// TwinCAT 3 PLC project plc_lfe_gem
// Title: LFE GEM
// Company: SLAC - LCLS
// ProjectVersion: 4.0.0
// ProgramVersion: 3.1.4022.4
// libraries:
//   LCLS General, * (SLAC)
//   LCLS Vacuum, * (SLAC - LCLS)
//   PMPS, * (SLAC - LCLS)
//   Tc2_ControllerToolbox, * (Beckhoff Automation GmbH)
//   Tc2_Standard, * (Beckhoff Automation GmbH)
//   Tc2_System, * (Beckhoff Automation GmbH)
//   Tc2_Utilities, * (Beckhoff Automation GmbH)
//   Tc3_Module, * (Beckhoff Automation GmbH)
// project tree:
//   DUTs/ E_PositionState.TcDUT, ST_MPA.TcDUT, ST_PressureSensor.TcDUT
//   Version/ Global_Version.TcGVL
//   GVLs/ GVL_Control.TcGVL, GVL_Devices.TcGVL, GVL_ILK.TcGVL, GVL_Sensors.TcGVL
//   / PlcTask.TcTTO
//   POUs/ DIAGNOSTICS.TcPOU, FB_MPA.TcPOU, FB_PressureSensor_PX219.TcPOU, FB_VGC_1.TcPOU, MAIN.TcPOU, PRG_GEM1_DIFF_PUMP.TcPOU, PRG_GEM2_DIFF_PUMP.TcPOU, PRG_GATT.TcPOU, PRG_GEM1.TcPOU, PRG_GEM2.TcPOU, PRG_ILK.TcPOU, PRG_PMPS.TcPOU, PRG_ROOTS.TcPOU, PRG_SATT.TcPOU, PRG_SENSORS.TcPOU
// real-time tasks:
//   TASK PlcTask: cycle T#10ms, priority 20, ADS port 350
// I/O:
//   DEVICE EMxL0 (EtherCAT), AmsNetId 172.21.88.32.4.1
//     PLC_EMxL0 (EK1200) [EK1200-5000 EtherCAT Power supply (2A E-Bus)]
//       PLC_EL_1 (EL2088) [EL2088 8Ch. Dig. Output 24V, 0.5A, switching to negative]
//       PLC_EL_2 (EL1088) [EL1088 8Ch. Dig. Input 24V, 3ms, negative]
//       PLC_EL_3 (EL1088) [EL1088 8Ch. Dig. Input 24V, 3ms, negative]
//       PLC_EL_4 (EL3064) [EL3064 4Ch. Ana. Input 0-10V]
//       PLC_EL_5 (EL3064) [EL3064 4Ch. Ana. Input 0-10V]
//       PLC_EL_6 (EL2088) [EL2088 8Ch. Dig. Output 24V, 0.5A, switching to negative]
//       PLC_EL_7 (EL1088) [EL1088 8Ch. Dig. Input 24V, 3ms, negative]
//       PLC_EL_8 (EL1088) [EL1088 8Ch. Dig. Input 24V, 3ms, negative]
//       PLC_EL_9 (EL9187) [EL9187 Potential Connection, 8 x Ground]
//       PLC_EL_10 (EL2088) [EL2088 8Ch. Dig. Output 24V, 0.5A, switching to negative]
//       PLC_EL_11 (EL1088) [EL1088 8Ch. Dig. Input 24V, 3ms, negative]
//       PLC_EL_12 (EL1088) [EL1088 8Ch. Dig. Input 24V, 3ms, negative]
//       PLC_EL_13 (EL2088) [EL2088 8Ch. Dig. Output 24V, 0.5A, switching to negative]
//       PLC_EL_14 (EL9187) [EL9187 Potential Connection, 8 x Ground]
//       PLC_EL_15 (EL6070) [EL6070 1Ch. Licensing-Terminal]
//       PMPS_FFO [EL2202 2Ch. Dig. Output 24V, 0.5A]
//       PMPS_PRE [EL6692 EtherCAT Bridge terminal (Primary)]
//       PLC_EK_18 (EK1110) [EK1110 EtherCAT extension]
//     DRL_MKS (EK1100) [EK1100 EtherCAT Coupler (2A E-Bus)]
//       MKS_E1 (EL3064) [EL3064 4Ch. Ana. Input 0-10V]
//       MKS_E2 (EL3064) [EL3064 4Ch. Ana. Input 0-10V]
//       MKS_E3 (EL2794) [EL2794 4Ch. Dig. Output 24V AC/DC, 2A, short-circuit-proof]
//       MKS_E4 (EL3064) [EL3064 4Ch. Ana. Input 0-10V]
//       MKS_E5 (EL3064) [EL3064 4Ch. Ana. Input 0-10V]
//       MKS_E6 (EL2794) [EL2794 4Ch. Dig. Output 24V AC/DC, 2A, short-circuit-proof]
//       MKS_E7 (EL3064) [EL3064 4Ch. Ana. Input 0-10V]
//       MKS_E8 (EL3064) [EL3064 4Ch. Ana. Input 0-10V]
//       MKS_E9 (EL2794) [EL2794 4Ch. Dig. Output 24V AC/DC, 2A, short-circuit-proof]
//       MKS_E10 (EL3064) [EL3064 4Ch. Ana. Input 0-10V]
//       MKS_E11 (EL3064) [EL3064 4Ch. Ana. Input 0-10V]
//       MKS_E12 (EL2794) [EL2794 4Ch. Dig. Output 24V AC/DC, 2A, short-circuit-proof]
//       MKS_E13 (EL3064) [EL3064 4Ch. Ana. Input 0-10V]
//       MKS_E14 (EL3064) [EL3064 4Ch. Ana. Input 0-10V]
//       MKS_E15 (EL2794) [EL2794 4Ch. Dig. Output 24V AC/DC, 2A, short-circuit-proof]
//       MKS_E16 (EK1110)
//     DRL_PTM (EK1100) [EK1100 EtherCAT Coupler (2A E-Bus)]
//       PTM_E1_EL1004
//       PTM_E2_EL1004 [EL1004 4Ch. Dig. Input 24V, 3ms]
//       PTM_E3_EL2798 [EL2798 8Ch. Dig. Output 24V AC/DC, 2A, potential-free]
//       PTM_E4_EL3064 [EL3064 4Ch. Ana. Input 0-10V]
//       PTM_E5_EL4004 [EL4004 4Ch. Ana. Output 0-10V, 12bit]
//       PTM_E6_EL3064 [EL3064 4Ch. Ana. Input 0-10V]
//       PTM_E7_EL2798 [EL2798 8Ch. Dig. Output 24V AC/DC, 2A, potential-free]
//       PTM_E8_EL1004 [EL1004 4Ch. Dig. Input 24V, 3ms]
//       PTM_E9_EL1004
//       PTM_E10_EL9410
//       PTM_E11_EL1004
//       PTM_E12_EL1004 [EL1004 4Ch. Dig. Input 24V, 3ms]
//       PTM_E13_EL2798 [EL2798 8Ch. Dig. Output 24V AC/DC, 2A, potential-free]
//       PTM_E14_EL3064
//       PTM_E15_EL4004 [EL4004 4Ch. Ana. Output 0-10V, 12bit]
//       PTM_E16_EL3064 [EL3064 4Ch. Ana. Input 0-10V]
//       PTM_E17_EL2798 [EL2798 8Ch. Dig. Output 24V AC/DC, 2A, potential-free]
//       PTM_E18_EL1004
//       PTM_E19_EL1004 [EL1004 4Ch. Dig. Input 24V, 3ms]
//       PTM_E20_EL2624 [EL2624 4Ch. Relay Output, NO (125V AC / 30V DC)]
//       PTM_E21_EL1088 [EL1088 8Ch. Dig. Input 24V, 3ms, negative]
//       PTM_E22_EL9187 [EL9187 Potential Connection, 8 x Ground]
//       PTM_E23_EL9011
//     L0S3_PNL_01_EB_1 (EP2338-0002) [EP2338-0002 8 Ch. Dig. Input/Output 24V, 0,5A, M12]
//     L0S3_PNL_01_EB_2 (EP2338-0002) [EP2338-0002 8 Ch. Dig. Input/Output 24V, 0,5A, M12]
//     L0S3_PNL_01_EB_3 (EP2338-0002) [EP2338-0002 8 Ch. Dig. Input/Output 24V, 0,5A, M12]
//     L0S3_PNL_01_EB_4 (EP2338-0002) [EP2338-0002 8 Ch. Dig. Input/Output 24V, 0,5A, M12]
//     L0S3_PNL_01_EB_5 (EP3174-0002) [EP3174-0002 4Ch. Ana. Input +/-10V, 0-10V, 0/4-20mA configurable]
//     L0S3_PNL_01_EB_6 (EP3174-0002) [EP3174-0002 4Ch. Ana. Input +/-10V, 0-10V, 0/4-20mA configurable]
//     L0S3_PNL_02_EB_1 (EP2338-0002) [EP2338-0002 8 Ch. Dig. Input/Output 24V, 0,5A, M12]
//     L0S3_PNL_02_EB_2 (EP2338-0002) [EP2338-0002 8 Ch. Dig. Input/Output 24V, 0,5A, M12]
//     L0S3_PNL_02_EB_3 (EP4374-0002) [EP4374-0002 2Ch. Ana. Input +/-10V, 0-10V, 0/4-20mA configurable; 2Ch. Ana. Output +/-10V, 0-10V, 0/4-20mA configurable]
//     L0S3_PNL_02_EB_4 (EP3174-0002) [EP3174-0002 4Ch. Ana. Input +/-10V, 0-10V, 0/4-20mA configurable]
//     L0S3_PNL_02_EB_5 (EP2624-0002) [EP2624-0002 4Ch. Relay Output, NO (125V AC / 30V DC)]
//     L0S3_PNL_03_EB_1 (EP2338-0002) [EP2338-0002 8 Ch. Dig. Input/Output 24V, 0,5A, M12]
//     L0S3_PNL_03_EB_2 (EP2338-0002) [EP2338-0002 8 Ch. Dig. Input/Output 24V, 0,5A, M12]
//     L0S3_PNL_03_EB_3 (EP2338-0002) [EP2338-0002 8 Ch. Dig. Input/Output 24V, 0,5A, M12]
//     L0S3_PNL_03_EB_4 (EP3174-0002) [EP3174-0002 4Ch. Ana. Input +/-10V, 0-10V, 0/4-20mA configurable]
//     L0S3_PNL_03_EB_5 (EP3174-0002) [EP3174-0002 4Ch. Ana. Input +/-10V, 0-10V, 0/4-20mA configurable]
//     L0S3_PNL_03_EB_6 (EP2624-0002) [EP2624-0002 4Ch. Relay Output, NO (125V AC / 30V DC)]
//     L0S3_PNL_03_EB_7 (EP2338-0002) [EP2338-0002 8 Ch. Dig. Input/Output 24V, 0,5A, M12]
//     L0S3_PNL_03_EB_8 (EP2624-0002) [EP2624-0002 4Ch. Relay Output, NO (125V AC / 30V DC)]
//     L0S3_PNL_03_EB_9 (EP2338-0002) [EP2338-0002 8 Ch. Dig. Input/Output 24V, 0,5A, M12]
//     L0S6_PNL_04_EB_1 (EP2338-0002) [EP2338-0002 8 Ch. Dig. Input/Output 24V, 0,5A, M12]
//     L0S6_PNL_04_EB_2 (EP3174-0002) [EP3174-0002 4Ch. Ana. Input +/-10V, 0-10V, 0/4-20mA configurable]
//     L0S6_PNL_04_EB_3 (EP4374-0002) [EP4374-0002 2Ch. Ana. Input +/-10V, 0-10V, 0/4-20mA configurable; 2Ch. Ana. Output +/-10V, 0-10V, 0/4-20mA configurable]
//     L0S6_PNL_04_EB_4 (EP2338-0002) [EP2338-0002 8 Ch. Dig. Input/Output 24V, 0,5A, M12]
//     L0S6_PNL_04_EB_5 (EP2338-0002) [EP2338-0002 8 Ch. Dig. Input/Output 24V, 0,5A, M12]
//     L0S6_PNL_04_EB_6 (EP2338-0002) [EP2338-0002 8 Ch. Dig. Input/Output 24V, 0,5A, M12]
//     L0S6_PNL_04_EB_7 (EP2338-0002) [EP2338-0002 8 Ch. Dig. Input/Output 24V, 0,5A, M12]
//     L0S6_PNL_04_EB_8 (EP2338-0002) [EP2338-0002 8 Ch. Dig. Input/Output 24V, 0,5A, M12]
//     L0S6_PNL_01_EB_1 (EP2338-0002) [EP2338-0002 8 Ch. Dig. Input/Output 24V, 0,5A, M12]
//     L0S6_PNL_01_EB_2 (EP2338-0002) [EP2338-0002 8 Ch. Dig. Input/Output 24V, 0,5A, M12]
//     L0S6_PNL_01_EB_3 (EP2338-0002) [EP2338-0002 8 Ch. Dig. Input/Output 24V, 0,5A, M12]
//     L0S6_PNL_01_EB_4 (EP3174-0002) [EP3174-0002 4Ch. Ana. Input +/-10V, 0-10V, 0/4-20mA configurable]
//     L0S6_PNL_01_EB_5 (EP3174-0002) [EP3174-0002 4Ch. Ana. Input +/-10V, 0-10V, 0/4-20mA configurable]
//     L0S6_PNL_01_EB_6 (EP2624-0002) [EP2624-0002 4Ch. Relay Output, NO (125V AC / 30V DC)]
//     L0S6_PNL_01_EB_7 (EP2338-0002) [EP2338-0002 8 Ch. Dig. Input/Output 24V, 0,5A, M12]
//     L0S6_PNL_01_EB_8 (EP2624-0002) [EP2624-0002 4Ch. Relay Output, NO (125V AC / 30V DC)]
//     L0S6_PNL_01_EB_9 (EP2338-0002) [EP2338-0002 8 Ch. Dig. Input/Output 24V, 0,5A, M12]
//     L0S6_PNL_02_EB_1 (EP2338-0002) [EP2338-0002 8 Ch. Dig. Input/Output 24V, 0,5A, M12]
//     L0S6_PNL_02_EB_2 (EP2338-0002) [EP2338-0002 8 Ch. Dig. Input/Output 24V, 0,5A, M12]
//     L0S6_PNL_02_EB_3 (EP4374-0002) [EP4374-0002 2Ch. Ana. Input +/-10V, 0-10V, 0/4-20mA configurable; 2Ch. Ana. Output +/-10V, 0-10V, 0/4-20mA configurable]
//     L0S6_PNL_02_EB_4 (EP3174-0002) [EP3174-0002 4Ch. Ana. Input +/-10V, 0-10V, 0/4-20mA configurable]
//     L0S6_PNL_02_EB_5 (EP2624-0002) [EP2624-0002 4Ch. Relay Output, NO (125V AC / 30V DC)]
//     L0S6_PNL_03_EB_1 (EP2338-0002) [EP2338-0002 8 Ch. Dig. Input/Output 24V, 0,5A, M12]
//     L0S6_PNL_03_EB_2 (EP2338-0002) [EP2338-0002 8 Ch. Dig. Input/Output 24V, 0,5A, M12]
//     L0S6_PNL_03_EB_3 (EP2338-0002) [EP2338-0002 8 Ch. Dig. Input/Output 24V, 0,5A, M12]
//     L0S6_PNL_03_EB_4 (EP2338-0002) [EP2338-0002 8 Ch. Dig. Input/Output 24V, 0,5A, M12]
//     L0S6_PNL_03_EB_5 (EP3174-0002) [EP3174-0002 4Ch. Ana. Input +/-10V, 0-10V, 0/4-20mA configurable]
//     L0S6_PNL_03_EB_6 (EP3174-0002) [EP3174-0002 4Ch. Ana. Input +/-10V, 0-10V, 0/4-20mA configurable]
// variable links:
//   plc_lfe_gem/plc_lfe_gem Instance <-> EMxL0 (EtherCAT)/DRL_MKS (EK1100)/MKS_E1 (EL3064)
//     PlcTask Inputs/GVL_Devices.GEM1_GCC_10.i_iPRESS_R <-> AI Standard Channel 1/Value
//     PlcTask Inputs/GVL_Devices.GEM1_GCC_20.i_iPRESS_R <-> AI Standard Channel 3/Value
//     PlcTask Inputs/GVL_Devices.GEM1_GPI_10.i_iPRESS_R <-> AI Standard Channel 4/Value
//   plc_lfe_gem/plc_lfe_gem Instance <-> EMxL0 (EtherCAT)/DRL_MKS (EK1100)/MKS_E10 (EL3064)
//     PlcTask Inputs/GVL_Devices.GEM2_GCC_50.i_iPRESS_R <-> AI Standard Channel 1/Value
//     PlcTask Inputs/GVL_Devices.GEM2_GCC_60.i_iPRESS_R <-> AI Standard Channel 3/Value
//     PlcTask Inputs/GVL_Devices.GEM2_GPI_50.i_iPRESS_R <-> AI Standard Channel 4/Value
//   plc_lfe_gem/plc_lfe_gem Instance <-> EMxL0 (EtherCAT)/DRL_MKS (EK1100)/MKS_E11 (EL3064)
//     PlcTask Inputs/GVL_Devices.GEM2_GPI_60.i_iPRESS_R <-> AI Standard Channel 1/Value
//   plc_lfe_gem/plc_lfe_gem Instance <-> EMxL0 (EtherCAT)/DRL_MKS (EK1100)/MKS_E12 (EL2794)
//     PlcTask Outputs/GVL_Devices.GEM2_GCC_50.q_xHV_DIS <-> Channel 1/Output
//     PlcTask Outputs/GVL_Devices.GEM2_GCC_60.q_xHV_DIS <-> Channel 2/Output
//   plc_lfe_gem/plc_lfe_gem Instance <-> EMxL0 (EtherCAT)/DRL_MKS (EK1100)/MKS_E13 (EL3064)
//     PlcTask Inputs/GVL_Devices.GEM2_GCC_70.i_iPRESS_R <-> AI Standard Channel 1/Value
//     PlcTask Inputs/GVL_Devices.GEM2_GPI_70.i_iPRESS_R <-> AI Standard Channel 4/Value
//   plc_lfe_gem/plc_lfe_gem Instance <-> EMxL0 (EtherCAT)/DRL_MKS (EK1100)/MKS_E14 (EL3064)
//     PlcTask Inputs/GVL_Devices.GEM1_GPI_60.i_iPRESS_R <-> AI Standard Channel 1/Value
//   plc_lfe_gem/plc_lfe_gem Instance <-> EMxL0 (EtherCAT)/DRL_MKS (EK1100)/MKS_E15 (EL2794)
//     PlcTask Outputs/GVL_Devices.GEM2_GCC_70.q_xHV_DIS <-> Channel 1/Output
//   plc_lfe_gem/plc_lfe_gem Instance <-> EMxL0 (EtherCAT)/DRL_MKS (EK1100)/MKS_E2 (EL3064)
//     PlcTask Inputs/GVL_Devices.GEM1_GPI_20.i_iPRESS_R <-> AI Standard Channel 1/Value
//   plc_lfe_gem/plc_lfe_gem Instance <-> EMxL0 (EtherCAT)/DRL_MKS (EK1100)/MKS_E3 (EL2794)
//     PlcTask Outputs/GVL_Devices.GEM1_GCC_10.q_xHV_DIS <-> Channel 1/Output
//     PlcTask Outputs/GVL_Devices.GEM1_GCC_20.q_xHV_DIS <-> Channel 2/Output
//   plc_lfe_gem/plc_lfe_gem Instance <-> EMxL0 (EtherCAT)/DRL_MKS (EK1100)/MKS_E4 (EL3064)
//     PlcTask Inputs/GVL_Devices.GEM1_GCC_30.i_iPRESS_R <-> AI Standard Channel 1/Value
//     PlcTask Inputs/GVL_Devices.GEM1_GCC_50.i_iPRESS_R <-> AI Standard Channel 3/Value
//     PlcTask Inputs/GVL_Devices.GEM1_GPI_30.i_iPRESS_R <-> AI Standard Channel 4/Value
//   plc_lfe_gem/plc_lfe_gem Instance <-> EMxL0 (EtherCAT)/DRL_MKS (EK1100)/MKS_E5 (EL3064)
//     PlcTask Inputs/GVL_Devices.GEM1_GPI_50.i_iPRESS_R <-> AI Standard Channel 1/Value
//   plc_lfe_gem/plc_lfe_gem Instance <-> EMxL0 (EtherCAT)/DRL_MKS (EK1100)/MKS_E6 (EL2794)
//     PlcTask Outputs/GVL_Devices.GEM1_GCC_30.q_xHV_DIS <-> Channel 1/Output
//     PlcTask Outputs/GVL_Devices.GEM1_GCC_50.q_xHV_DIS <-> Channel 2/Output
//   plc_lfe_gem/plc_lfe_gem Instance <-> EMxL0 (EtherCAT)/DRL_MKS (EK1100)/MKS_E7 (EL3064)
//     PlcTask Inputs/GVL_Devices.GATT_GPI_10.i_iPRESS_R <-> AI Standard Channel 2/Value
//     PlcTask Inputs/GVL_Devices.GEM2_GCC_30.i_iPRESS_R <-> AI Standard Channel 1/Value
//     PlcTask Inputs/GVL_Devices.GEM2_GPI_10.i_iPRESS_R <-> AI Standard Channel 4/Value
//     PlcTask Inputs/GVL_Devices.GEM2_GPI_30.i_iPRESS_R <-> AI Standard Channel 3/Value
//   plc_lfe_gem/plc_lfe_gem Instance <-> EMxL0 (EtherCAT)/DRL_MKS (EK1100)/MKS_E9 (EL2794)
//     PlcTask Outputs/GVL_Devices.GEM2_GCC_30.q_xHV_DIS <-> Channel 1/Output
//   plc_lfe_gem/plc_lfe_gem Instance <-> EMxL0 (EtherCAT)/DRL_PTM (EK1100)/PTM_E11_EL1004
//     PlcTask Inputs/GVL_Devices.GEM2_PTM_30.i_xAtSpd <-> Channel 2/Input
//     PlcTask Inputs/GVL_Devices.GEM2_PTM_30.i_xDecel <-> Channel 1/Input
//     PlcTask Inputs/GVL_Devices.GEM2_PTM_30.i_xNCFault <-> Channel 3/Input
//     PlcTask Inputs/GVL_Devices.GEM2_PTM_30.i_xRotate <-> Channel 4/Input
//   plc_lfe_gem/plc_lfe_gem Instance <-> EMxL0 (EtherCAT)/DRL_PTM (EK1100)/PTM_E12_EL1004
//     PlcTask Inputs/GVL_Devices.GEM2_PTM_30.i_xAccel <-> Channel 1/Input
//   plc_lfe_gem/plc_lfe_gem Instance <-> EMxL0 (EtherCAT)/DRL_PTM (EK1100)/PTM_E13_EL2798
//     PlcTask Outputs/GVL_Devices.GEM2_PTM_30.q_xProtection <-> Channel 4/Output
//     PlcTask Outputs/GVL_Devices.GEM2_PTM_30.q_xReset <-> Channel 1/Output
//     PlcTask Outputs/GVL_Devices.GEM2_PTM_30.q_xSetSpeed <-> Channel 5/Output
//     PlcTask Outputs/GVL_Devices.GEM2_PTM_30.q_xStart <-> Channel 2/Output
//     PlcTask Outputs/GVL_Devices.GEM2_PTM_30.q_xStop <-> Channel 3/Output
//   plc_lfe_gem/plc_lfe_gem Instance <-> EMxL0 (EtherCAT)/DRL_PTM (EK1100)/PTM_E14_EL3064
//     PlcTask Inputs/GVL_Devices.GEM2_PTM_30.i_iCurrentMon <-> AI Standard Channel 2/Value
//     PlcTask Inputs/GVL_Devices.GEM2_PTM_30.i_iRawSpeed <-> AI Standard Channel 1/Value
//     PlcTask Inputs/GVL_Devices.GEM2_PTM_30.i_iTempMon <-> AI Standard Channel 3/Value
//   plc_lfe_gem/plc_lfe_gem Instance <-> EMxL0 (EtherCAT)/DRL_PTM (EK1100)/PTM_E15_EL4004
//     PlcTask Outputs/GVL_Devices.GEM2_PTM_30.q_iSpeedSet <-> AO Outputs Channel 1/Analog output
//     PlcTask Outputs/GVL_Devices.GEM2_PTM_50.q_iSpeedSet <-> AO Outputs Channel 3/Analog output
//   plc_lfe_gem/plc_lfe_gem Instance <-> EMxL0 (EtherCAT)/DRL_PTM (EK1100)/PTM_E16_EL3064
//     PlcTask Inputs/GVL_Devices.GEM2_PTM_50.i_iCurrentMon <-> AI Standard Channel 2/Value
//     PlcTask Inputs/GVL_Devices.GEM2_PTM_50.i_iRawSpeed <-> AI Standard Channel 1/Value
//     PlcTask Inputs/GVL_Devices.GEM2_PTM_50.i_iTempMon <-> AI Standard Channel 3/Value
//   plc_lfe_gem/plc_lfe_gem Instance <-> EMxL0 (EtherCAT)/DRL_PTM (EK1100)/PTM_E17_EL2798
//     PlcTask Outputs/GVL_Devices.GEM2_PTM_50.q_xProtection <-> Channel 4/Output
//     PlcTask Outputs/GVL_Devices.GEM2_PTM_50.q_xReset <-> Channel 1/Output
//     PlcTask Outputs/GVL_Devices.GEM2_PTM_50.q_xSetSpeed <-> Channel 5/Output
//     PlcTask Outputs/GVL_Devices.GEM2_PTM_50.q_xStart <-> Channel 2/Output
//     PlcTask Outputs/GVL_Devices.GEM2_PTM_50.q_xStop <-> Channel 3/Output
//   plc_lfe_gem/plc_lfe_gem Instance <-> EMxL0 (EtherCAT)/DRL_PTM (EK1100)/PTM_E18_EL1004
//     PlcTask Inputs/GVL_Devices.GEM2_PTM_50.i_xAtSpd <-> Channel 2/Input
//     PlcTask Inputs/GVL_Devices.GEM2_PTM_50.i_xDecel <-> Channel 1/Input
//     PlcTask Inputs/GVL_Devices.GEM2_PTM_50.i_xNCFault <-> Channel 3/Input
//     PlcTask Inputs/GVL_Devices.GEM2_PTM_50.i_xRotate <-> Channel 4/Input
//   plc_lfe_gem/plc_lfe_gem Instance <-> EMxL0 (EtherCAT)/DRL_PTM (EK1100)/PTM_E19_EL1004
//     PlcTask Inputs/GVL_Devices.GEM2_PTM_50.i_xAccel <-> Channel 1/Input
//   plc_lfe_gem/plc_lfe_gem Instance <-> EMxL0 (EtherCAT)/DRL_PTM (EK1100)/PTM_E1_EL1004
//     PlcTask Inputs/GVL_Devices.GEM1_PTM_30.i_xAtSpd <-> Channel 2/Input
//     PlcTask Inputs/GVL_Devices.GEM1_PTM_30.i_xDecel <-> Channel 1/Input
//     PlcTask Inputs/GVL_Devices.GEM1_PTM_30.i_xNCFault <-> Channel 3/Input
//     PlcTask Inputs/GVL_Devices.GEM1_PTM_30.i_xRotate <-> Channel 4/Input
//   plc_lfe_gem/plc_lfe_gem Instance <-> EMxL0 (EtherCAT)/DRL_PTM (EK1100)/PTM_E20_EL2624
//     PlcTask Outputs/GVL_Devices.GEM1_PTM_10.q_RunDO <-> Channel 1/Output
//     PlcTask Outputs/GVL_Devices.GEM1_PTM_20.q_RunDO <-> Channel 2/Output
//     PlcTask Outputs/GVL_Devices.GEM2_PTM_60.q_RunDO <-> Channel 3/Output
//     PlcTask Outputs/GVL_Devices.GEM2_PTM_70.q_RunDO <-> Channel 4/Output
//   plc_lfe_gem/plc_lfe_gem Instance <-> EMxL0 (EtherCAT)/DRL_PTM (EK1100)/PTM_E21_EL1088
//     PlcTask Inputs/GVL_Devices.GEM1_PTM_10.i_xAtSpd <-> Channel 1/Input
//     PlcTask Inputs/GVL_Devices.GEM1_PTM_20.i_xAtSpd <-> Channel 3/Input
//     PlcTask Inputs/GVL_Devices.GEM2_PTM_60.i_xAtSpd <-> Channel 5/Input
//     PlcTask Inputs/GVL_Devices.GEM2_PTM_70.i_xAtSpd <-> Channel 7/Input
//     PlcTask Inputs/GVL_Devices.GEM1_PTM_10.i_xFault <-> Channel 2/Input
//     PlcTask Inputs/GVL_Devices.GEM1_PTM_20.i_xFault <-> Channel 4/Input
//     PlcTask Inputs/GVL_Devices.GEM2_PTM_60.i_xFault <-> Channel 6/Input
//     PlcTask Inputs/GVL_Devices.GEM2_PTM_70.i_xFault <-> Channel 8/Input
//   plc_lfe_gem/plc_lfe_gem Instance <-> EMxL0 (EtherCAT)/DRL_PTM (EK1100)/PTM_E2_EL1004
//     PlcTask Inputs/GVL_Devices.GEM1_PTM_30.i_xAccel <-> Channel 1/Input
//   plc_lfe_gem/plc_lfe_gem Instance <-> EMxL0 (EtherCAT)/DRL_PTM (EK1100)/PTM_E3_EL2798
//     PlcTask Outputs/GVL_Devices.GEM1_PTM_30.q_xProtection <-> Channel 4/Output
//     PlcTask Outputs/GVL_Devices.GEM1_PTM_30.q_xReset <-> Channel 1/Output
//     PlcTask Outputs/GVL_Devices.GEM1_PTM_30.q_xSetSpeed <-> Channel 5/Output
//     PlcTask Outputs/GVL_Devices.GEM1_PTM_30.q_xStart <-> Channel 2/Output
//     PlcTask Outputs/GVL_Devices.GEM1_PTM_30.q_xStop <-> Channel 3/Output
//   plc_lfe_gem/plc_lfe_gem Instance <-> EMxL0 (EtherCAT)/DRL_PTM (EK1100)/PTM_E4_EL3064
//     PlcTask Inputs/GVL_Devices.GEM1_PTM_30.i_iCurrentMon <-> AI Standard Channel 2/Value
//     PlcTask Inputs/GVL_Devices.GEM1_PTM_30.i_iRawSpeed <-> AI Standard Channel 1/Value
//     PlcTask Inputs/GVL_Devices.GEM1_PTM_30.i_iTempMon <-> AI Standard Channel 3/Value
//   plc_lfe_gem/plc_lfe_gem Instance <-> EMxL0 (EtherCAT)/DRL_PTM (EK1100)/PTM_E5_EL4004
//     PlcTask Outputs/GVL_Devices.GEM1_PTM_30.q_iSpeedSet <-> AO Outputs Channel 1/Analog output
//     PlcTask Outputs/GVL_Devices.GEM1_PTM_50.q_iSpeedSet <-> AO Outputs Channel 3/Analog output
//   plc_lfe_gem/plc_lfe_gem Instance <-> EMxL0 (EtherCAT)/DRL_PTM (EK1100)/PTM_E6_EL3064
//     PlcTask Inputs/GVL_Devices.GEM1_PTM_50.i_iCurrentMon <-> AI Standard Channel 2/Value
//     PlcTask Inputs/GVL_Devices.GEM1_PTM_50.i_iRawSpeed <-> AI Standard Channel 1/Value
//     PlcTask Inputs/GVL_Devices.GEM1_PTM_50.i_iTempMon <-> AI Standard Channel 3/Value
//   plc_lfe_gem/plc_lfe_gem Instance <-> EMxL0 (EtherCAT)/DRL_PTM (EK1100)/PTM_E7_EL2798
//     PlcTask Outputs/GVL_Devices.GEM1_PTM_50.q_xProtection <-> Channel 4/Output
//     PlcTask Outputs/GVL_Devices.GEM1_PTM_50.q_xReset <-> Channel 1/Output
//     PlcTask Outputs/GVL_Devices.GEM1_PTM_50.q_xSetSpeed <-> Channel 5/Output
//     PlcTask Outputs/GVL_Devices.GEM1_PTM_50.q_xStart <-> Channel 2/Output
//     PlcTask Outputs/GVL_Devices.GEM1_PTM_50.q_xStop <-> Channel 3/Output
//   plc_lfe_gem/plc_lfe_gem Instance <-> EMxL0 (EtherCAT)/DRL_PTM (EK1100)/PTM_E8_EL1004
//     PlcTask Inputs/GVL_Devices.GEM1_PTM_50.i_xAtSpd <-> Channel 2/Input
//     PlcTask Inputs/GVL_Devices.GEM1_PTM_50.i_xDecel <-> Channel 1/Input
//     PlcTask Inputs/GVL_Devices.GEM1_PTM_50.i_xNCFault <-> Channel 3/Input
//     PlcTask Inputs/GVL_Devices.GEM1_PTM_50.i_xRotate <-> Channel 4/Input
//   plc_lfe_gem/plc_lfe_gem Instance <-> EMxL0 (EtherCAT)/DRL_PTM (EK1100)/PTM_E9_EL1004
//     PlcTask Inputs/GVL_Devices.GEM1_PTM_50.i_xAccel <-> Channel 1/Input
//   plc_lfe_gem/plc_lfe_gem Instance <-> EMxL0 (EtherCAT)/L0S3_PNL_01_EB_1 (EP2338-0002)
//     PlcTask Inputs/GVL_Devices.GEM1_VGC_10.i_xClsLS <-> Channel 2/Input
//     PlcTask Inputs/GVL_Devices.GEM1_VGC_10.i_xOpnLS <-> Channel 1/Input
//     PlcTask Inputs/GVL_Devices.GEM1_VRC_10.i_xClsLS <-> Channel 6/Input
//     PlcTask Inputs/GVL_Devices.GEM1_VRC_10.i_xOpnLS <-> Channel 5/Input
//     PlcTask Outputs/GVL_Devices.GEM1_VGC_10.q_xOPN_DO <-> Channel 11/Output
//     PlcTask Outputs/GVL_Devices.GEM1_VRC_10.q_xOPN_DO <-> Channel 15/Output
//   plc_lfe_gem/plc_lfe_gem Instance <-> EMxL0 (EtherCAT)/L0S3_PNL_01_EB_2 (EP2338-0002)
//     PlcTask Inputs/GVL_Devices.GEM1_VGC_20.i_xClsLS <-> Channel 2/Input
//     PlcTask Inputs/GVL_Devices.GEM1_VGC_30.i_xClsLS <-> Channel 6/Input
//     PlcTask Inputs/GVL_Devices.GEM1_VGC_20.i_xOpnLS <-> Channel 1/Input
//     PlcTask Inputs/GVL_Devices.GEM1_VGC_30.i_xOpnLS <-> Channel 5/Input
//     PlcTask Outputs/GVL_Devices.GEM1_VGC_20.q_xOPN_DO <-> Channel 11/Output
//     PlcTask Outputs/GVL_Devices.GEM1_VGC_30.q_xOPN_DO <-> Channel 15/Output
//   plc_lfe_gem/plc_lfe_gem Instance <-> EMxL0 (EtherCAT)/L0S3_PNL_01_EB_3 (EP2338-0002)
//     PlcTask Inputs/GVL_Devices.GEM1_VRC_20.i_xClsLS <-> Channel 6/Input
//     PlcTask Inputs/GVL_Devices.GEM1_VRC_20.i_xOpnLS <-> Channel 5/Input
//     PlcTask Outputs/GVL_Devices.GEM1_VRC_20.q_xOPN_DO <-> Channel 15/Output
//     PlcTask Outputs/GVL_Devices.GEM1_VVC_20.q_xCLS_DO <-> Channel 11/Output
//   plc_lfe_gem/plc_lfe_gem Instance <-> EMxL0 (EtherCAT)/L0S3_PNL_01_EB_4 (EP2338-0002)
//     PlcTask Inputs/GVL_Devices.GEM1_VRC_30.i_xClsLS <-> Channel 6/Input
//     PlcTask Inputs/GVL_Devices.GEM1_VRC_30.i_xOpnLS <-> Channel 5/Input
//     PlcTask Outputs/GVL_Devices.GEM1_VRC_30.q_xOPN_DO <-> Channel 15/Output
//     PlcTask Outputs/GVL_Devices.GEM1_VVC_30.q_xCLS_DO <-> Channel 11/Output
//   plc_lfe_gem/plc_lfe_gem Instance <-> EMxL0 (EtherCAT)/L0S3_PNL_01_EB_5 (EP3174-0002)
//     PlcTask Inputs/GVL_Devices.GEM1_GPI_11.i_iPRESS_R <-> AI Standard Channel 3/Value
//     PlcTask Inputs/GVL_Devices.GEM1_GPI_31.i_iPRESS_R <-> AI Standard Channel 4/Value
//   plc_lfe_gem/plc_lfe_gem Instance <-> EMxL0 (EtherCAT)/L0S3_PNL_02_EB_1 (EP2338-0002)
//     PlcTask Inputs/GVL_Devices.GEM1_VGC_40.i_xClsLS <-> Channel 2/Input
//     PlcTask Inputs/GVL_Devices.GEM1_VGC_50.i_xClsLS <-> Channel 6/Input
//     PlcTask Inputs/GVL_Devices.GEM1_VGC_40.i_xOpnLS <-> Channel 1/Input
//     PlcTask Inputs/GVL_Devices.GEM1_VGC_50.i_xOpnLS <-> Channel 5/Input
//     PlcTask Outputs/GVL_Devices.GEM1_VGC_40.q_xOPN_DO <-> Channel 11/Output
//     PlcTask Outputs/GVL_Devices.GEM1_VGC_50.q_xOPN_DO <-> Channel 15/Output
//   plc_lfe_gem/plc_lfe_gem Instance <-> EMxL0 (EtherCAT)/L0S3_PNL_02_EB_2 (EP2338-0002)
//     PlcTask Outputs/GVL_Devices.GEM1_VVC_40.q_xOPN_DO <-> Channel 15/Output
//   plc_lfe_gem/plc_lfe_gem Instance <-> EMxL0 (EtherCAT)/L0S3_PNL_02_EB_3 (EP4374-0002)
//     PlcTask Outputs/GVL_Devices.GEM1_VCN_40.q_iRawPosition <-> AO Outputs Channel 4/Analog output
//   plc_lfe_gem/plc_lfe_gem Instance <-> EMxL0 (EtherCAT)/L0S3_PNL_02_EB_4 (EP3174-0002)
//     PlcTask Inputs/GVL_Devices.GEM1_GCM_41.i_iPRESS_R <-> AI Standard Channel 1/Value
//     PlcTask Inputs/GVL_Devices.GEM1_GCM_42.i_iPRESS_R <-> AI Standard Channel 2/Value
//   plc_lfe_gem/plc_lfe_gem Instance <-> EMxL0 (EtherCAT)/L0S3_PNL_03_EB_1 (EP2338-0002)
//     PlcTask Inputs/GVL_Devices.GEM1_VGC_60.i_xClsLS <-> Channel 6/Input
//     PlcTask Inputs/GVL_Devices.GEM1_VGC_60.i_xOpnLS <-> Channel 5/Input
//     PlcTask Inputs/GVL_Devices.GEM1_VRC_50.i_xClsLS <-> Channel 2/Input
//     PlcTask Inputs/GVL_Devices.GEM1_VRC_50.i_xOpnLS <-> Channel 1/Input
//     PlcTask Outputs/GVL_Devices.GEM1_VGC_60.q_xOPN_DO <-> Channel 15/Output
//     PlcTask Outputs/GVL_Devices.GEM1_VRC_50.q_xOPN_DO <-> Channel 11/Output
//   plc_lfe_gem/plc_lfe_gem Instance <-> EMxL0 (EtherCAT)/L0S3_PNL_03_EB_2 (EP2338-0002)
//     PlcTask Inputs/GVL_Devices.GEM1_VRC_60.i_xClsLS <-> Channel 6/Input
//     PlcTask Inputs/GVL_Devices.GEM1_VRC_60.i_xOpnLS <-> Channel 5/Input
//     PlcTask Outputs/GVL_Devices.GEM1_VRC_60.q_xOPN_DO <-> Channel 15/Output
//     PlcTask Outputs/GVL_Devices.GEM1_VVC_50.q_xCLS_DO <-> Channel 11/Output
//   plc_lfe_gem/plc_lfe_gem Instance <-> EMxL0 (EtherCAT)/L0S3_PNL_03_EB_3 (EP2338-0002)
//     PlcTask Inputs/GVL_Devices.GEM1_VGC_70.i_xClsLS <-> Channel 2/Input
//     PlcTask Inputs/GVL_Devices.GEM1_VGC_70.i_xOpnLS <-> Channel 1/Input
//     PlcTask Inputs/GVL_Devices.GEM1_VRC_70.i_xClsLS <-> Channel 6/Input
//     PlcTask Inputs/GVL_Devices.GEM1_VRC_70.i_xOpnLS <-> Channel 5/Input
//     PlcTask Outputs/GVL_Devices.GEM1_VGC_70.q_xOPN_DO <-> Channel 11/Output
//     PlcTask Outputs/GVL_Devices.GEM1_VRC_70.q_xOPN_DO <-> Channel 15/Output
//   plc_lfe_gem/plc_lfe_gem Instance <-> EMxL0 (EtherCAT)/L0S3_PNL_03_EB_4 (EP3174-0002)
//     PlcTask Inputs/GVL_Devices.GEM1_GPI_51.i_iPRESS_R <-> AI Standard Channel 3/Value
//   plc_lfe_gem/plc_lfe_gem Instance <-> EMxL0 (EtherCAT)/L0S3_PNL_03_EB_5 (EP3174-0002)
//     PlcTask Inputs/GVL_Devices.GEM1_GPI_61.i_iPRESS_R <-> AI Standard Channel 2/Value
//     PlcTask Inputs/GVL_Devices.GEM1_GPI_71.i_iPRESS_R <-> AI Standard Channel 3/Value
//   plc_lfe_gem/plc_lfe_gem Instance <-> EMxL0 (EtherCAT)/L0S3_PNL_03_EB_6 (EP2624-0002)
//     PlcTask Outputs/GVL_Devices.GEM1_PRO_60.q_xLspdDo <-> Channel 2/Output
//     PlcTask Outputs/GVL_Devices.GEM1_PRO_60.q_xResetDo <-> Channel 3/Output
//     PlcTask Outputs/GVL_Devices.GEM1_PRO_60.q_xRunDO <-> Channel 1/Output
//   plc_lfe_gem/plc_lfe_gem Instance <-> EMxL0 (EtherCAT)/L0S3_PNL_03_EB_7 (EP2338-0002)
//     PlcTask Inputs/GVL_Devices.GEM1_PRO_60.i_xAlarm <-> Channel 6/Input
//     PlcTask Inputs/GVL_Devices.GEM1_PRO_60.i_xIsRun <-> Channel 1/Input
//     PlcTask Inputs/GVL_Devices.GEM1_PRO_60.i_xWarning <-> Channel 5/Input
//     PlcTask Outputs/GVL_Devices.GEM1_PRO_20.q_xRunDo <-> Channel 11/Output
//     PlcTask Outputs/GVL_Devices.GEM1_PRO_30.q_xRunDo <-> Channel 12/Output
//     PlcTask Outputs/GVL_Devices.GEM1_PRO_50.q_xRunDo <-> Channel 15/Output
//   plc_lfe_gem/plc_lfe_gem Instance <-> EMxL0 (EtherCAT)/L0S3_PNL_03_EB_8 (EP2624-0002)
//     PlcTask Outputs/GVL_Devices.GEM1_PRO_70.q_xLspdDo <-> Channel 2/Output
//     PlcTask Outputs/GVL_Devices.GEM1_PRO_70.q_xResetDo <-> Channel 3/Output
//     PlcTask Outputs/GVL_Devices.GEM1_PRO_70.q_xRunDO <-> Channel 1/Output
//   plc_lfe_gem/plc_lfe_gem Instance <-> EMxL0 (EtherCAT)/L0S3_PNL_03_EB_9 (EP2338-0002)
//     PlcTask Inputs/GVL_Devices.GEM1_PRO_70.i_xAlarm <-> Channel 6/Input
//     PlcTask Inputs/GVL_Devices.GEM1_PRO_70.i_xIsRun <-> Channel 1/Input
//     PlcTask Inputs/GVL_Devices.GEM1_PRO_70.i_xWarning <-> Channel 5/Input
//   plc_lfe_gem/plc_lfe_gem Instance <-> EMxL0 (EtherCAT)/L0S6_PNL_01_EB_1 (EP2338-0002)
//     PlcTask Inputs/GVL_Devices.GEM2_VGC_10.i_xClsLS <-> Channel 2/Input
//     PlcTask Inputs/GVL_Devices.GEM2_VGC_20.i_xClsLS <-> Channel 6/Input
//     PlcTask Inputs/GVL_Devices.GEM2_VGC_10.i_xOpnLS <-> Channel 1/Input
//     PlcTask Inputs/GVL_Devices.GEM2_VGC_20.i_xOpnLS <-> Channel 5/Input
//     PlcTask Outputs/GVL_Devices.GEM2_VGC_10.q_xOPN_DO <-> Channel 11/Output
//     PlcTask Outputs/GVL_Devices.GEM2_VGC_20.q_xOPN_DO <-> Channel 15/Output
//   plc_lfe_gem/plc_lfe_gem Instance <-> EMxL0 (EtherCAT)/L0S6_PNL_01_EB_2 (EP2338-0002)
//     PlcTask Inputs/GVL_Devices.GEM2_VRC_10.i_xClsLS <-> Channel 2/Input
//     PlcTask Inputs/GVL_Devices.GEM2_VRC_20.i_xClsLS <-> Channel 6/Input
//     PlcTask Inputs/GVL_Devices.GEM2_VRC_10.i_xOpnLS <-> Channel 1/Input
//     PlcTask Inputs/GVL_Devices.GEM2_VRC_20.i_xOpnLS <-> Channel 5/Input
//     PlcTask Outputs/GVL_Devices.GEM2_VRC_10.q_xOPN_DO <-> Channel 11/Output
//     PlcTask Outputs/GVL_Devices.GEM2_VRC_20.q_xOPN_DO <-> Channel 15/Output
//   plc_lfe_gem/plc_lfe_gem Instance <-> EMxL0 (EtherCAT)/L0S6_PNL_01_EB_3 (EP2338-0002)
//     PlcTask Inputs/GVL_Devices.GEM2_VRC_30.i_xClsLS <-> Channel 2/Input
//     PlcTask Inputs/GVL_Devices.GEM2_VRC_30.i_xOpnLS <-> Channel 1/Input
//     PlcTask Outputs/GVL_Devices.GEM2_VRC_30.q_xOPN_DO <-> Channel 11/Output
//     PlcTask Outputs/GVL_Devices.GEM2_VVC_30.q_xCLS_DO <-> Channel 15/Output
//   plc_lfe_gem/plc_lfe_gem Instance <-> EMxL0 (EtherCAT)/L0S6_PNL_01_EB_4 (EP3174-0002)
//     PlcTask Inputs/GVL_Devices.GEM2_GPI_11.i_iPRESS_R <-> AI Standard Channel 2/Value
//     PlcTask Inputs/GVL_Devices.GEM2_GPI_21.i_iPRESS_R <-> AI Standard Channel 3/Value
//     PlcTask Inputs/GVL_Devices.GEM2_GPI_31.i_iPRESS_R <-> AI Standard Channel 4/Value
//   plc_lfe_gem/plc_lfe_gem Instance <-> EMxL0 (EtherCAT)/L0S6_PNL_01_EB_6 (EP2624-0002)
//     PlcTask Outputs/GVL_Devices.GEM2_PRO_10.q_xLspdDo <-> Channel 2/Output
//     PlcTask Outputs/GVL_Devices.GEM2_PRO_10.q_xResetDo <-> Channel 3/Output
//     PlcTask Outputs/GVL_Devices.GEM2_PRO_10.q_xRunDO <-> Channel 1/Output
//   plc_lfe_gem/plc_lfe_gem Instance <-> EMxL0 (EtherCAT)/L0S6_PNL_01_EB_7 (EP2338-0002)
//     PlcTask Inputs/GVL_Devices.GEM2_PRO_10.i_xAlarm <-> Channel 6/Input
//     PlcTask Inputs/GVL_Devices.GEM2_PRO_10.i_xIsRun <-> Channel 1/Input
//     PlcTask Inputs/GVL_Devices.GEM2_PRO_10.i_xWarning <-> Channel 5/Input
//     PlcTask Outputs/GVL_Devices.GEM2_PRO_30.q_xRunDo <-> Channel 11/Output
//     PlcTask Outputs/GVL_Devices.GEM2_PRO_50.q_xRunDo <-> Channel 12/Output
//     PlcTask Outputs/GVL_Devices.GEM2_PRO_60.q_xRunDo <-> Channel 15/Output
//   plc_lfe_gem/plc_lfe_gem Instance <-> EMxL0 (EtherCAT)/L0S6_PNL_01_EB_8 (EP2624-0002)
//     PlcTask Outputs/GVL_Devices.GEM2_PRO_20.q_xLspdDo <-> Channel 2/Output
//     PlcTask Outputs/GVL_Devices.GEM2_PRO_20.q_xResetDo <-> Channel 3/Output
//     PlcTask Outputs/GVL_Devices.GEM2_PRO_20.q_xRunDO <-> Channel 1/Output
//   plc_lfe_gem/plc_lfe_gem Instance <-> EMxL0 (EtherCAT)/L0S6_PNL_01_EB_9 (EP2338-0002)
//     PlcTask Inputs/GVL_Devices.GEM2_PRO_20.i_xAlarm <-> Channel 6/Input
//     PlcTask Inputs/GVL_Devices.GEM2_PRO_20.i_xIsRun <-> Channel 1/Input
//     PlcTask Inputs/GVL_Devices.GEM2_PRO_20.i_xWarning <-> Channel 5/Input
//   plc_lfe_gem/plc_lfe_gem Instance <-> EMxL0 (EtherCAT)/L0S6_PNL_02_EB_1 (EP2338-0002)
//     PlcTask Inputs/GVL_Devices.GEM2_VGC_30.i_xClsLS <-> Channel 2/Input
//     PlcTask Inputs/GVL_Devices.GEM2_VGC_40.i_xClsLS <-> Channel 6/Input
//     PlcTask Inputs/GVL_Devices.GEM2_VGC_30.i_xOpnLS <-> Channel 1/Input
//     PlcTask Inputs/GVL_Devices.GEM2_VGC_40.i_xOpnLS <-> Channel 5/Input
//     PlcTask Outputs/GVL_Devices.GEM2_VGC_30.q_xOPN_DO <-> Channel 11/Output
//     PlcTask Outputs/GVL_Devices.GEM2_VGC_40.q_xOPN_DO <-> Channel 15/Output
//   plc_lfe_gem/plc_lfe_gem Instance <-> EMxL0 (EtherCAT)/L0S6_PNL_02_EB_2 (EP2338-0002)
//     PlcTask Outputs/GVL_Devices.GEM2_VVC_40.q_xOPN_DO <-> Channel 15/Output
//   plc_lfe_gem/plc_lfe_gem Instance <-> EMxL0 (EtherCAT)/L0S6_PNL_02_EB_3 (EP4374-0002)
//     PlcTask Outputs/GVL_Devices.GEM2_VCN_40.q_iRawPosition <-> AO Outputs Channel 4/Analog output
//   plc_lfe_gem/plc_lfe_gem Instance <-> EMxL0 (EtherCAT)/L0S6_PNL_02_EB_4 (EP3174-0002)
//     PlcTask Inputs/GVL_Devices.GEM2_GCM_41.i_iPRESS_R <-> AI Standard Channel 1/Value
//     PlcTask Inputs/GVL_Devices.GEM2_GCM_42.i_iPRESS_R <-> AI Standard Channel 2/Value
//   plc_lfe_gem/plc_lfe_gem Instance <-> EMxL0 (EtherCAT)/L0S6_PNL_03_EB_1 (EP2338-0002)
//     PlcTask Inputs/GVL_Devices.GEM2_VGC_50.i_xClsLS <-> Channel 2/Input
//     PlcTask Inputs/GVL_Devices.GEM2_VGC_50.i_xOpnLS <-> Channel 1/Input
//     PlcTask Inputs/GVL_Devices.GEM2_VRC_50.i_xClsLS <-> Channel 6/Input
//     PlcTask Inputs/GVL_Devices.GEM2_VRC_50.i_xOpnLS <-> Channel 5/Input
//     PlcTask Outputs/GVL_Devices.GEM2_VGC_50.q_xOPN_DO <-> Channel 11/Output
//     PlcTask Outputs/GVL_Devices.GEM2_VRC_50.q_xOPN_DO <-> Channel 15/Output
//   plc_lfe_gem/plc_lfe_gem Instance <-> EMxL0 (EtherCAT)/L0S6_PNL_03_EB_2 (EP2338-0002)
//     PlcTask Inputs/GVL_Devices.GEM2_VRC_60.i_xClsLS <-> Channel 2/Input
//     PlcTask Inputs/GVL_Devices.GEM2_VRC_70.i_xClsLS <-> Channel 6/Input
//     PlcTask Inputs/GVL_Devices.GEM2_VRC_60.i_xOpnLS <-> Channel 1/Input
//     PlcTask Inputs/GVL_Devices.GEM2_VRC_70.i_xOpnLS <-> Channel 5/Input
//     PlcTask Outputs/GVL_Devices.GEM2_VRC_60.q_xOPN_DO <-> Channel 11/Output
//     PlcTask Outputs/GVL_Devices.GEM2_VRC_70.q_xOPN_DO <-> Channel 15/Output
//   plc_lfe_gem/plc_lfe_gem Instance <-> EMxL0 (EtherCAT)/L0S6_PNL_03_EB_3 (EP2338-0002)
//     PlcTask Inputs/GVL_Devices.GEM2_VGC_60.i_xClsLS <-> Channel 2/Input
//     PlcTask Inputs/GVL_Devices.GEM2_VGC_70.i_xClsLS <-> Channel 6/Input
//     PlcTask Inputs/GVL_Devices.GEM2_VGC_60.i_xOpnLS <-> Channel 1/Input
//     PlcTask Inputs/GVL_Devices.GEM2_VGC_70.i_xOpnLS <-> Channel 5/Input
//     PlcTask Outputs/GVL_Devices.GEM2_VGC_60.q_xOPN_DO <-> Channel 11/Output
//     PlcTask Outputs/GVL_Devices.GEM2_VGC_70.q_xOPN_DO <-> Channel 15/Output
//   plc_lfe_gem/plc_lfe_gem Instance <-> EMxL0 (EtherCAT)/L0S6_PNL_03_EB_4 (EP2338-0002)
//     PlcTask Outputs/GVL_Devices.GEM2_VVC_50.q_xCLS_DO <-> Channel 15/Output
//     PlcTask Outputs/GVL_Devices.GEM2_VVC_70.q_xCLS_DO <-> Channel 16/Output
//   plc_lfe_gem/plc_lfe_gem Instance <-> EMxL0 (EtherCAT)/L0S6_PNL_03_EB_6 (EP3174-0002)
//     PlcTask Inputs/GVL_Devices.GEM2_GPI_51.i_iPRESS_R <-> AI Standard Channel 2/Value
//     PlcTask Inputs/GVL_Devices.GEM2_GPI_61.i_iPRESS_R <-> AI Standard Channel 1/Value
//   plc_lfe_gem/plc_lfe_gem Instance <-> EMxL0 (EtherCAT)/L0S6_PNL_04_EB_1 (EP2338-0002)
//     PlcTask Inputs/GVL_Devices.GATT_VRC_10.i_xClsLS <-> Channel 2/Input
//     PlcTask Inputs/GVL_Devices.GATT_VRC_10.i_xOpnLS <-> Channel 1/Input
//     PlcTask Outputs/GVL_Devices.GATT_VRC_10.q_xOPN_DO <-> Channel 11/Output
//     PlcTask Outputs/GVL_Devices.GATT_VVC_10.q_xOPN_DO <-> Channel 15/Output
//   plc_lfe_gem/plc_lfe_gem Instance <-> EMxL0 (EtherCAT)/L0S6_PNL_04_EB_2 (EP3174-0002)
//     PlcTask Inputs/GVL_Devices.GATT_GMP_10.i_iPRESS_R <-> AI Standard Channel 2/Value
//   plc_lfe_gem/plc_lfe_gem Instance <-> EMxL0 (EtherCAT)/L0S6_PNL_04_EB_3 (EP4374-0002)
//     PlcTask Inputs/GVL_Devices.GATT_GMP_11.i_iPRESS_R <-> AI Inputs Channel 1/Value
//   plc_lfe_gem/plc_lfe_gem Instance <-> EMxL0 (EtherCAT)/PLC_EMxL0 (EK1200)/PMPS_FFO
//     PlcTask Outputs/GVL_ILK.g_FastFaultOutput1.q_xFastFaultOut <-> Channel 1/Output
//     PlcTask Outputs/GVL_ILK.g_FastFaultOutput2.q_xFastFaultOut <-> Channel 2/Output
//   plc_lfe_gem/plc_lfe_gem Instance <-> EMxL0 (EtherCAT)/PLC_EMxL0 (EK1200)/PMPS_PRE
//     PlcTask Inputs/PRG_PMPS.fbArbiterIO.i_stCurrentBP <-> IO Inputs/CurrentBP
//     PlcTask Inputs/PRG_PMPS.fbArbiterIO.xTxPDO_state <-> SYNC Inputs/TxPDO state
//     PlcTask Inputs/PRG_PMPS.fbArbiterIO.xTxPDO_toggle <-> SYNC Inputs/TxPDO toggle
//     PlcTask Outputs/PRG_PMPS.fbArbiterIO.q_stRequestedBP <-> IO Outputs/RequestedBP

CONFIGURATION plc_lfe_gem
    RESOURCE PLC ON TwinCAT3
        TASK PlcTask(INTERVAL := T#10ms, PRIORITY := 20);
        PROGRAM MAIN WITH PlcTask : MAIN;
    END_RESOURCE
END_CONFIGURATION

// ---- DUTs/E_PositionState.TcDUT
{attribute 'qualified_only'}
{attribute 'strict'}
TYPE E_PositionState :
(
RETRACTED	:= 0,
INSERTED	:= 1,
MOVING	:= 2,
INVALID :=3
);
END_TYPE

// ---- DUTs/ST_MPA.TcDUT
TYPE ST_MPA :
STRUCT
    //Readbacks
    {attribute 'pytmc' := '
    pv: IN;
    io: i;
    '}
    i_bInLS	:	BOOL;
    {attribute 'pytmc' := '
    pv: OUT;
    io: i;
    '}
    i_bOutLS	:	BOOL;
    //Controls
    {attribute 'pytmc' := '
    pv: INSERT_DO;
    io: i;
    '}
    q_bRetract	:	BOOL;
    {attribute 'pytmc' := '
    pv: RETRACT_DO;
    io: i;
    '}
    q_bInsert	:	BOOL;
//    q_xRetract_Do : Bool;


    //Logic and supervisory
    {attribute 'pytmc' := '
    pv: ILKOK;
    io: i;
    '}
    bILK_OK: BOOL;
    {attribute 'pytmc' := '
    pv: INSERT_OK;
    io: i;
    '}
    bInsertOK	:	BOOL;
    {attribute 'pytmc' := '
    pv: RETRACT_OK;
    io: i;
    '}
    bRetractOK	:	BOOL;
    {attribute 'pytmc' := '
    pv: IN_CMD;
    io: io;
    '}
    bInsert_SW		:	BOOL;
    {attribute 'pytmc' := '
    pv: OUT_CMD;
    io: io;
    '}
    bRetract_SW	:	BOOL;
    {attribute 'pytmc' := '
    pv: ERROR;
    io: io;
    '}
    bErrorPresent : BOOL;
    {attribute 'pytmc' := '
    pv: POS_STATE ;
    type: mbbi ;
    field: ZRST RETRACTED ;
    field: ONST INSERTED ;
    field: TWST MOVING ;
    field: THST INVALID ;
    io: i
    '}

    eState	:	E_PositionState := E_PositionState.INVALID;

END_STRUCT
END_TYPE

// ---- DUTs/ST_PressureSensor.TcDUT
TYPE ST_PressureSensor :
STRUCT
    {attribute 'pytmc' := '
    pv: PRESS;
    io: i;
    '}
    rPRESS: REAL; //This is the human-readable pressure
    {attribute 'pytmc' := '
    pv: iPRESS;
    io: i;
    '}
    iPRESS_R : INT ; //input pressure in machine form
    {attribute 'pytmc' := '
    pv: PRESS_SP;
    io: io;
    '}
    rPressSP: REAL ; // EPICS Pressure setpoint
    {attribute 'pytmc' := '
    pv: MIN_SP;
    io: io;
    '}
    rMinPressSP : REAL;  // Low limit of pressure setpoint
    {attribute 'pytmc' := '
    pv: MAX_SP;
    io: io;
    '}
    rMaxPressSP : REAL;	// High limit of pressure setpoint
    {attribute 'pytmc' := '
    pv: SCALE;
    io: io;
    '}
    rFULL_SCALE: REAL; // Full scale
    {attribute 'pytmc' := '
    pv: ALARM;
    field: ZNAM Normal;
    field: ONAM Alarm;
    io: i;
    '}
    xPstateAlarm : BOOL; // 0:Normal, 1:Alarm


END_STRUCT
END_TYPE

// ---- Version/Global_Version.TcGVL
{attribute 'TcGenerated'}
{attribute 'no-analysis'}
{attribute 'linkalways'}
// This function has been automatically generated from the project information.
VAR_GLOBAL CONSTANT
    {attribute 'const_non_replaced'}
    stLibVersion_LFE_GEM : ST_LibVersion := (iMajor := 4, iMinor := 0, iBuild := 0, iRevision := 0, nFlags := 1, sVersion := '4.0.0');
END_VAR

// ---- GVLs/GVL_Control.TcGVL
VAR_GLOBAL
    {attribute 'pytmc' :=' pv: EM1L0:GEM:CNTRL:SP;
    field: HOPR 1000;
    field: LOPR 0;
    field: PREC 2;
    field: EGU "TORR";
    '}
    fGEM1SetpointValue : REAL:=0;
    {attribute 'pytmc' :=' pv: EM2L0:GEM:CNTRL:SP;
    field: HOPR 1000;
    field: LOPR 0;
    field: PREC 2;
    field: EGU "TORR";
    '}
    fGEM2SetpointValue : REAL:=0;


    {attribute 'pytmc' :=' pv: EM1L0:GEM:CNTRL:GO;
      field: ZNAM STOP;
     field: ONAM START;
     io: io;
     '}
    GEM1_GO : BOOL:=false;

    {attribute 'pytmc' :=' pv: EM2L0:GEM:CNTRL:GO;
     field: ZNAM STOP;
     field: ONAM START;
     io: io; '}
    GEM2_GO : BOOL:=false;
END_VAR

// ---- GVLs/GVL_Devices.TcGVL
VAR_GLOBAL

    (*Upstream Interface*)
    (*Gauges*)
    USG_PIN: FB_TPIP_ADS;
    USG_GCC: FB_TGCC_ADS;
    DSG_PIN: FB_TPIP_ADS;
    (*Valves*)
    DSV_VGC: FB_Valve_Interface;

    iWatchdog:UDINT;//The watchdog variable name written to by the remote plc


(*EM1L0*)
(*Gauges*)
    {attribute 'pytmc' :=' pv: EM1L0:GEM:GCC:10 '}
    {attribute 'TcLinkTo' := 	'.i_iPRESS_R	:=	TIIB[MKS_E1 (EL3064)]^AI Standard Channel 1^Value;
                                 .q_xHV_DIS		:= 	TIIB[MKS_E3 (EL2794)]^Channel 1^Output'}
    GEM1_GCC_10 : FB_MKS422;

    {attribute 'pytmc' :=' pv: EM1L0:GEM:GPI:10 '}
    {attribute 'TcLinkTo' := 	'.i_iPRESS_R	:=	TIIB[MKS_E1 (EL3064)]^AI Standard Channel 4^Value'}
    GEM1_GPI_10 : FB_MKS317A;

    {attribute 'pytmc' :=' pv: EM1L0:GEM:GCC:20 '}
    {attribute 'TcLinkTo' := 	'.i_iPRESS_R	:=	TIIB[MKS_E1 (EL3064)]^AI Standard Channel 3^Value;
                                 .q_xHV_DIS		:= 	TIIB[MKS_E3 (EL2794)]^Channel 2^Output'}
    GEM1_GCC_20 : FB_MKS422;

    {attribute 'pytmc' :=' pv: EM1L0:GEM:GPI:20 '}
    {attribute 'TcLinkTo' := 	'.i_iPRESS_R	:=	TIIB[MKS_E2 (EL3064)]^AI Standard Channel 1^Value'}
    GEM1_GPI_20 : FB_MKS317A;

    {attribute 'pytmc' :=' pv: EM1L0:GEM:GCC:30 '}
    {attribute 'TcLinkTo' := 	'.i_iPRESS_R	:=	TIIB[MKS_E4 (EL3064)]^AI Standard Channel 1^Value;
                                 .q_xHV_DIS		:= 	TIIB[MKS_E6 (EL2794)]^Channel 1^Output'}
    GEM1_GCC_30 : FB_MKS422;

    {attribute 'pytmc' :=' pv: EM1L0:GEM:GPI:30 '}
    {attribute 'TcLinkTo' := 	'.i_iPRESS_R	:=	TIIB[MKS_E4 (EL3064)]^AI Standard Channel 4^Value'}
    GEM1_GPI_30 : FB_MKS317A;

    {attribute 'pytmc' :=' pv: EM1L0:GEM:GCC:50 '}
    {attribute 'TcLinkTo' := 	'.i_iPRESS_R	:=	TIIB[MKS_E4 (EL3064)]^AI Standard Channel 3^Value;
                                 .q_xHV_DIS		:= 	TIIB[MKS_E6 (EL2794)]^Channel 2^Output'}
    GEM1_GCC_50 : FB_MKS422;

    {attribute 'pytmc' :=' pv: EM1L0:GEM:GPI:50 '}
    {attribute 'TcLinkTo' := 	'.i_iPRESS_R	:=	TIIB[MKS_E5 (EL3064)]^AI Standard Channel 1^Value'}
    GEM1_GPI_50 : FB_MKS317A;

    {attribute 'pytmc' :=' pv: EM1L0:GEM:GPI:11 '}
    {attribute 'TcLinkTo' := 	'.i_iPRESS_R	:=	TIIB[L0S3_PNL_01_EB_5 (EP3174-0002)]^AI Standard Channel 3^Value'}
    GEM1_GPI_11 : FB_MKS275;

    {attribute 'pytmc' :=' pv: EM1L0:GEM:GPI:31 '}
    {attribute 'TcLinkTo' := 	'.i_iPRESS_R	:=	TIIB[L0S3_PNL_01_EB_5 (EP3174-0002)]^AI Standard Channel 4^Value'}
    GEM1_GPI_31 : FB_MKS275;

    {attribute 'pytmc' :=' pv: EM1L0:GEM:GPI:51 '}
    {attribute 'TcLinkTo' := 	'.i_iPRESS_R	:=	TIIB[L0S3_PNL_03_EB_4 (EP3174-0002)]^AI Standard Channel 3^Value'}
    GEM1_GPI_51 : FB_MKS275;

    {attribute 'pytmc' :=' pv: EM1L0:GEM:GPI:60 '}
    {attribute 'TcLinkTo' := 	'.i_iPRESS_R	:=	TIIB[MKS_E14 (EL3064)]^AI Standard Channel 1^Value'}
    GEM1_GPI_60 : FB_MKS317A;

    {attribute 'pytmc' :=' pv: EM1L0:GEM:GPI:61 '}
    {attribute 'TcLinkTo' := 	'.i_iPRESS_R	:=	TIIB[L0S3_PNL_03_EB_5 (EP3174-0002)]^AI Standard Channel 2^Value'}
    GEM1_GPI_61 : FB_MKS275;

    {attribute 'pytmc' :=' pv: EM1L0:GEM:GPI:71 '}
    {attribute 'TcLinkTo' := 	'.i_iPRESS_R	:=	TIIB[L0S3_PNL_03_EB_5 (EP3174-0002)]^AI Standard Channel 3^Value'}
    GEM1_GPI_71 : FB_MKS275;

(*detector*)
    {attribute 'pytmc' :=' pv: EM1L0:GEM:GCM:41 '}
    {attribute 'TcLinkTo' := 	'.i_iPRESS_R	:=	TIIB[L0S3_PNL_02_EB_4 (EP3174-0002)]^AI Standard Channel 1^Value'}
    GEM1_GCM_41 : FB_GCM;
    {attribute 'pytmc' :=' pv: EM1L0:GEM:GCM:42 '}
    {attribute 'TcLinkTo' := 	'.i_iPRESS_R	:=	TIIB[L0S3_PNL_02_EB_4 (EP3174-0002)]^AI Standard Channel 2^Value'}
    GEM1_GCM_42 : FB_GCM;
    (*Pseudo gauge device Structure to combine the readings of two GCM gauges*)
    {attribute 'pytmc' :=' pv: EM1L0:GEM:GCM:40 '}
    GEM1_GCM_40 : ST_VG;
(* N2 cutt off valve *)
    {attribute 'pytmc' :=' pv: EM1L0:GEM:VVC:40'}
    {attribute 'TcLinkTo' := 	'.q_xOPN_DO	:=	TIIB[L0S3_PNL_02_EB_2 (EP2338-0002)]^Channel 15^Output'}
    GEM1_VVC_40: FB_VVC;
(*Pressure Control valve*)
    {attribute 'pytmc' :=' pv: EM1L0:GEM:VCN:40 '}
    {attribute 'TcLinkTo' := 	'.q_iRawPosition	:=	TIIB[L0S3_PNL_02_EB_3 (EP4374-0002)]^AO Outputs Channel 4^Analog output'}
    GEM1_VCN_40 : FB_VCN;

(* aperture valves*)
    {attribute 'pytmc' :=' pv: EM1L0:GEM:VGC:10 '}
    {attribute 'TcLinkTo' := 	'.i_xOpnLS	:=	TIIB[L0S3_PNL_01_EB_1 (EP2338-0002)]^Channel 1^Input;
                                 .i_xClsLS	:=	TIIB[L0S3_PNL_01_EB_1 (EP2338-0002)]^Channel 2^Input;
                                 .q_xOPN_DO	:=	TIIB[L0S3_PNL_01_EB_1 (EP2338-0002)]^Channel 11^Output'}
    GEM1_VGC_10: FB_VGC;

    {attribute 'pytmc' :=' pv: EM1L0:GEM:VGC:20 '}
    {attribute 'TcLinkTo' := 	'.i_xOpnLS	:=	TIIB[L0S3_PNL_01_EB_2 (EP2338-0002)]^Channel 1^Input;
                                 .i_xClsLS	:=	TIIB[L0S3_PNL_01_EB_2 (EP2338-0002)]^Channel 2^Input;
                                 .q_xOPN_DO	:=	TIIB[L0S3_PNL_01_EB_2 (EP2338-0002)]^Channel 11^Output'}
    GEM1_VGC_20: FB_VGC;

    {attribute 'pytmc' :=' pv: EM1L0:GEM:VGC:30 '}
    {attribute 'TcLinkTo' := 	'.i_xOpnLS	:=	TIIB[L0S3_PNL_01_EB_2 (EP2338-0002)]^Channel 5^Input;
                                 .i_xClsLS	:=	TIIB[L0S3_PNL_01_EB_2 (EP2338-0002)]^Channel 6^Input;
                                 .q_xOPN_DO	:=	TIIB[L0S3_PNL_01_EB_2 (EP2338-0002)]^Channel 15^Output'}
    GEM1_VGC_30: FB_VGC;

    {attribute 'pytmc' :=' pv: EM1L0:GEM:VGC:40 '}
    {attribute 'TcLinkTo' := 	'.i_xOpnLS	:=	TIIB[L0S3_PNL_02_EB_1 (EP2338-0002)]^Channel 1^Input;
                                 .i_xClsLS	:=	TIIB[L0S3_PNL_02_EB_1 (EP2338-0002)]^Channel 2^Input;
                                 .q_xOPN_DO	:=	TIIB[L0S3_PNL_02_EB_1 (EP2338-0002)]^Channel 11^Output'}
    GEM1_VGC_40: FB_VGC;

    {attribute 'pytmc' :=' pv: EM1L0:GEM:VGC:50 '}
    {attribute 'TcLinkTo' := 	'.i_xOpnLS	:=	TIIB[L0S3_PNL_02_EB_1 (EP2338-0002)]^Channel 5^Input;
                                 .i_xClsLS	:=	TIIB[L0S3_PNL_02_EB_1 (EP2338-0002)]^Channel 6^Input;
                                 .q_xOPN_DO	:=	TIIB[L0S3_PNL_02_EB_1 (EP2338-0002)]^Channel 15^Output'}
    GEM1_VGC_50: FB_VGC;

    {attribute 'pytmc' :=' pv: EM1L0:GEM:VGC:60 '}
    {attribute 'TcLinkTo' := 	'.i_xOpnLS	:=	TIIB[L0S3_PNL_03_EB_1 (EP2338-0002)]^Channel 5^Input;
                                 .i_xClsLS	:=	TIIB[L0S3_PNL_03_EB_1 (EP2338-0002)]^Channel 6^Input;
                                 .q_xOPN_DO	:=	TIIB[L0S3_PNL_03_EB_1 (EP2338-0002)]^Channel 15^Output'}
    GEM1_VGC_60: FB_VGC;

    {attribute 'pytmc' :=' pv: EM1L0:GEM:VGC:70 '}
    {attribute 'TcLinkTo' := 	'.i_xOpnLS	:=	TIIB[L0S3_PNL_03_EB_3 (EP2338-0002)]^Channel 1^Input;
                                 .i_xClsLS	:=	TIIB[L0S3_PNL_03_EB_3 (EP2338-0002)]^Channel 2^Input;
                                 .q_xOPN_DO	:=	TIIB[L0S3_PNL_03_EB_3 (EP2338-0002)]^Channel 11^Output'}
    GEM1_VGC_70: FB_VGC;

(*Turbo Isolation valves*)
    {attribute 'pytmc' :=' pv: EM1L0:GEM:VRC:10 '}
    {attribute 'TcLinkTo' := 	'.i_xOpnLS	:=	TIIB[L0S3_PNL_01_EB_1 (EP2338-0002)]^Channel 5^Input;
                                 .i_xClsLS	:=	TIIB[L0S3_PNL_01_EB_1 (EP2338-0002)]^Channel 6^Input;
                                 .q_xOPN_DO	:=	TIIB[L0S3_PNL_01_EB_1 (EP2338-0002)]^Channel 15^Output'}
    GEM1_VRC_10: FB_VRC;

    {attribute 'pytmc' :=' pv: EM1L0:GEM:VRC:20 '}
    {attribute 'TcLinkTo' := 	'.i_xOpnLS	:=	TIIB[L0S3_PNL_01_EB_3 (EP2338-0002)]^Channel 5^Input;
                                 .i_xClsLS	:=	TIIB[L0S3_PNL_01_EB_3 (EP2338-0002)]^Channel 6^Input;
                                 .q_xOPN_DO	:=	TIIB[L0S3_PNL_01_EB_3 (EP2338-0002)]^Channel 15^Output'}
    GEM1_VRC_20: FB_VRC;

    {attribute 'pytmc' :=' pv: EM1L0:GEM:VRC:30 '}
    {attribute 'TcLinkTo' := 	'.i_xOpnLS	:=	TIIB[L0S3_PNL_01_EB_4 (EP2338-0002)]^Channel 5^Input;
                                 .i_xClsLS	:=	TIIB[L0S3_PNL_01_EB_4 (EP2338-0002)]^Channel 6^Input;
                                 .q_xOPN_DO	:=	TIIB[L0S3_PNL_01_EB_4 (EP2338-0002)]^Channel 15^Output'}
    GEM1_VRC_30: FB_VRC;

    {attribute 'pytmc' :=' pv: EM1L0:GEM:VRC:50 '}
    {attribute 'TcLinkTo' := 	'.i_xOpnLS	:=	TIIB[L0S3_PNL_03_EB_1 (EP2338-0002)]^Channel 1^Input;
                                 .i_xClsLS	:=	TIIB[L0S3_PNL_03_EB_1 (EP2338-0002)]^Channel 2^Input;
                                 .q_xOPN_DO	:=	TIIB[L0S3_PNL_03_EB_1 (EP2338-0002)]^Channel 11^Output'}
    GEM1_VRC_50: FB_VRC;

(*Kashiyama Valves*)
    {attribute 'pytmc' :=' pv: EM1L0:GEM:VRC:60 '}
    {attribute 'TcLinkTo' := 	'.i_xOpnLS	:=	TIIB[L0S3_PNL_03_EB_2 (EP2338-0002)]^Channel 5^Input;
                                 .i_xClsLS	:=	TIIB[L0S3_PNL_03_EB_2 (EP2338-0002)]^Channel 6^Input;
                                 .q_xOPN_DO	:=	TIIB[L0S3_PNL_03_EB_2 (EP2338-0002)]^Channel 15^Output'}
    GEM1_VRC_60:FB_Kashiyama_VRC;

    {attribute 'pytmc' :=' pv: EM1L0:GEM:VRC:70 '}
    {attribute 'TcLinkTo' := 	'.i_xOpnLS	:=	TIIB[L0S3_PNL_03_EB_3 (EP2338-0002)]^Channel 5^Input;
                                 .i_xClsLS	:=	TIIB[L0S3_PNL_03_EB_3 (EP2338-0002)]^Channel 6^Input;
                                 .q_xOPN_DO	:=	TIIB[L0S3_PNL_03_EB_3 (EP2338-0002)]^Channel 15^Output'}
    GEM1_VRC_70:FB_Kashiyama_VRC;

(*Kashiyama pumps*)

    {attribute 'pytmc' :=' pv: EM1L0:GEM:PRO:60 '}
    {attribute 'TcLinkTo' := 	'.i_xIsRun	:=	TIIB[L0S3_PNL_03_EB_7 (EP2338-0002)]^Channel 1^Input;
                                 .i_xLocal	:=	TIIB[L0S3_PNL_03_EB_7 (EP2338-0002)]^Channel 2^Input;
                                 .i_xWarning :=	TIIB[L0S3_PNL_03_EB_7 (EP2338-0002)]^Channel 5^Input;
                                 .i_xAlarm :=	TIIB[L0S3_PNL_03_EB_7 (EP2338-0002)]^Channel 6^Input;
                                 .q_xRunDO	:=	TIIB[L0S3_PNL_03_EB_6 (EP2624-0002)]^Channel 1^Output;
                                 .q_xLspdDo	:=	TIIB[L0S3_PNL_03_EB_6 (EP2624-0002)]^Channel 2^Output;
                                 .q_xResetDo:=	TIIB[L0S3_PNL_03_EB_6 (EP2624-0002)]^Channel 3^Output'}
    GEM1_PRO_60: FB_KashiyamaPump;

    {attribute 'pytmc' :=' pv: EM1L0:GEM:PRO:70 '}
    {attribute 'TcLinkTo' := 	'.i_xIsRun	:=	TIIB[L0S3_PNL_03_EB_9 (EP2338-0002)]^Channel 1^Input;
                                 .i_xLocal	:=	TIIB[L0S3_PNL_03_EB_9 (EP2338-0002)]^Channel 2^Input;
                                 .i_xWarning :=	TIIB[L0S3_PNL_03_EB_9 (EP2338-0002)]^Channel 5^Input;
                                 .i_xAlarm :=	TIIB[L0S3_PNL_03_EB_9 (EP2338-0002)]^Channel 6^Input;
                                 .q_xRunDO	:=	TIIB[L0S3_PNL_03_EB_8 (EP2624-0002)]^Channel 1^Output;
                                 .q_xLspdDo	:=	TIIB[L0S3_PNL_03_EB_8 (EP2624-0002)]^Channel 2^Output;
                                 .q_xResetDo:=	TIIB[L0S3_PNL_03_EB_8 (EP2624-0002)]^Channel 3^Output'}
    GEM1_PRO_70: FB_KashiyamaPump;

(*Turbos*)
    (*{attribute 'pytmc' :=' pv: EM1L0:GEM:PTM:10 '}
    {attribute 'TcLinkTo' := 	'.i_xR1	:=	TIIB[PLC_EL_2 (EL1088)]^Channel 1^Input;
                                 .i_xLSpd :=	TIIB[PLC_EL_2 (EL1088)]^Channel 2^Input;
                                 .i_xSTART	:=	TIIB[PLC_EL_2 (EL1088)]^Channel 3^Input;
                                 .i_xFault	:=	TIIB[PLC_EL_2 (EL1088)]^Channel 4^Input;
                                 .i_iPowerMon := TIIB[PLC_EL_4 (EL3064)]^AI Standard Channel 1^Value;
                                 .q_RunDO	:=	TIIB[PLC_EL_1 (EL2088)]^Channel 1^Output'}
    GEM1_PTM_10 : FB_PTM_Agilent;*)

    {attribute 'pytmc' :=' pv: EM1L0:GEM:PTM:10 '}
    {attribute 'TcLinkTo' := 	'.i_xAtSpd	:=	TIIB[PTM_E21_EL1088]^Channel 1^Input;
                                 .i_xFault :=	TIIB[PTM_E21_EL1088]^Channel 2^Input;
                                 .q_RunDO	:=	TIIB[PTM_E20_EL2624]^Channel 1^Output'}
    GEM1_PTM_10 : FB_PTM_TwisTorr;
    (*{attribute 'pytmc' :=' pv: EM1L0:GEM:PTM:20 '}
    {attribute 'TcLinkTo' := 	'.i_xR1	:=	TIIB[PLC_EL_2 (EL1088)]^Channel 5^Input;
                                 .i_xLSpd :=	TIIB[PLC_EL_2 (EL1088)]^Channel 6^Input;
                                 .i_xSTART	:=	TIIB[PLC_EL_2 (EL1088)]^Channel 7^Input;
                                 .i_xFault	:=	TIIB[PLC_EL_2 (EL1088)]^Channel 8^Input;
                                 .i_iPowerMon := TIIB[PLC_EL_4 (EL3064)]^AI Standard Channel 2^Value;
                                 .q_RunDO	:=	TIIB[PLC_EL_1 (EL2088)]^Channel 2^Output'}
    GEM1_PTM_20 : FB_PTM_Agilent;*)

    {attribute 'pytmc' :=' pv: EM1L0:GEM:PTM:20 '}
    {attribute 'TcLinkTo' := 	'.i_xAtSpd	:=	TIIB[PTM_E21_EL1088]^Channel 3^Input;
                                 .i_xFault :=	TIIB[PTM_E21_EL1088]^Channel 4^Input;
                                 .q_RunDO	:=	TIIB[PTM_E20_EL2624]^Channel 2^Output'}
    GEM1_PTM_20 : FB_PTM_TwisTorr;

    {attribute 'pytmc' :=' pv: EM1L0:GEM:PTM:30 '}
    {attribute 'TcLinkTo' := 	'.i_xDecel	:=	TIIB[PTM_E1_EL1004]^Channel 1^Input;
                                 .i_xAtSpd	:=	TIIB[PTM_E1_EL1004]^Channel 2^Input;
                                 .i_xNCFault :=	TIIB[PTM_E1_EL1004]^Channel 3^Input;
                                 .i_xRotate	:=	TIIB[PTM_E1_EL1004]^Channel 4^Input;
                                 .i_xAccel :=	TIIB[PTM_E2_EL1004]^Channel 1^Input;
                                 .i_iRawSpeed := TIIB[PTM_E4_EL3064]^AI Standard Channel 1^Value;
                                 .i_iCurrentMon := TIIB[PTM_E4_EL3064]^AI Standard Channel 2^Value;
                                 .i_iTempMon := TIIB[PTM_E4_EL3064]^AI Standard Channel 3^Value;
                                 .q_xReset	:=	TIIB[PTM_E3_EL2798]^Channel 1^Output;
                                 .q_xStart	:=	TIIB[PTM_E3_EL2798]^Channel 2^Output;
                                 .q_xStop	:=	TIIB[PTM_E3_EL2798]^Channel 3^Output;
                                 .q_xProtection	:=	TIIB[PTM_E3_EL2798]^Channel 4^Output;
                                 .q_xSetSpeed	:=	TIIB[PTM_E3_EL2798]^Channel 5^Output;
                                 .q_iSpeedSet	:=	TIIB[PTM_E5_EL4004]^AO Outputs Channel 1^Analog output'}
    GEM1_PTM_30 : FB_PTM_Ebara_010M;
    (*{attribute 'pytmc' :=' pv: EM1L0:GEM:PTM:50 '} REMOVE
    {attribute 'TcLinkTo' := 	'.i_xR1	:=	TIIB[PLC_EL_3 (EL1088)]^Channel 5^Input;
                                 .i_xLSpd :=	TIIB[PLC_EL_3 (EL1088)]^Channel 6^Input;
                                 .i_xSTART	:=	TIIB[PLC_EL_3 (EL1088)]^Channel 7^Input;
                                 .i_xFault	:=	TIIB[PLC_EL_3 (EL1088)]^Channel 8^Input;
                                 .i_iCurrentMon := TIIB[PLC_EL_4 (EL3064)]^AI Standard Channel 4^Value;
                                 .q_RunDO	:=	TIIB[PLC_EL_1 (EL2088)]^Channel 4^Output'}
    GEM1_PTM_50 : FB_PTM_Agilent;*)

    {attribute 'pytmc' :=' pv: EM1L0:GEM:PTM:50 '}
    {attribute 'TcLinkTo' := 	'.i_xDecel	:=	TIIB[PTM_E8_EL1004]^Channel 1^Input;
                                 .i_xAtSpd	:=	TIIB[PTM_E8_EL1004]^Channel 2^Input;
                                 .i_xNCFault :=	TIIB[PTM_E8_EL1004]^Channel 3^Input;
                                 .i_xRotate	:=	TIIB[PTM_E8_EL1004]^Channel 4^Input;
                                 .i_xAccel :=	TIIB[PTM_E9_EL1004]^Channel 1^Input;
                                 .i_iRawSpeed := TIIB[PTM_E6_EL3064]^AI Standard Channel 1^Value;
                                 .i_iCurrentMon := TIIB[PTM_E6_EL3064]^AI Standard Channel 2^Value;
                                 .i_iTempMon := TIIB[PTM_E6_EL3064]^AI Standard Channel 3^Value;
                                 .q_xReset	:=	TIIB[PTM_E7_EL2798]^Channel 1^Output;
                                 .q_xStart	:=	TIIB[PTM_E7_EL2798]^Channel 2^Output;
                                 .q_xStop	:=	TIIB[PTM_E7_EL2798]^Channel 3^Output;
                                 .q_xProtection	:=	TIIB[PTM_E7_EL2798]^Channel 4^Output;
                                 .q_xSetSpeed	:=	TIIB[PTM_E7_EL2798]^Channel 5^Output;
                                 .q_iSpeedSet	:=	TIIB[PTM_E5_EL4004]^AO Outputs Channel 3^Analog output'}
    GEM1_PTM_50 : FB_PTM_Ebara_010M;


(*Turbo vent valves*) (*deprecated*)
    {attribute 'pytmc' :=' pv: EM1L0:GEM:VVC:20 '}
    {attribute 'TcLinkTo' := 	'.q_xCLS_DO	:=	TIIB[L0S3_PNL_01_EB_3 (EP2338-0002)]^Channel 11^Output'}
    GEM1_VVC_20: FB_TurbVentvalve_NO;
    {attribute 'pytmc' :=' pv: EM1L0:GEM:VVC:30 '}
    {attribute 'TcLinkTo' := 	'.q_xCLS_DO	:=	TIIB[L0S3_PNL_01_EB_4 (EP2338-0002)]^Channel 11^Output'}
    GEM1_VVC_30: FB_TurbVentvalve_NO;
    {attribute 'pytmc' :=' pv: EM1L0:GEM:VVC:50 '}
    {attribute 'TcLinkTo' := 	'.q_xCLS_DO	:=	TIIB[L0S3_PNL_03_EB_2 (EP2338-0002)]^Channel 11^Output'}
    GEM1_VVC_50: FB_TurbVentvalve_NO;

(*Scroll Pumps*)
    {attribute 'pytmc' :=' pv: EM1L0:GEM:PRO:20 '}
    {attribute 'TcLinkTo' := 	'.q_xRunDo	:=	TIIB[L0S3_PNL_03_EB_7 (EP2338-0002)]^Channel 11^Output'}
    GEM1_PRO_20 : FB_ScrollPump;
    {attribute 'pytmc' :=' pv: EM1L0:GEM:PRO:30 '}
    {attribute 'TcLinkTo' := 	'.q_xRunDo	:=	TIIB[L0S3_PNL_03_EB_7 (EP2338-0002)]^Channel 12^Output'}
    GEM1_PRO_30 : FB_ScrollPump;
    {attribute 'pytmc' :=' pv: EM1L0:GEM:PRO:50 '}
    {attribute 'TcLinkTo' := 	'.q_xRunDo	:=	TIIB[L0S3_PNL_03_EB_7 (EP2338-0002)]^Channel 15^Output'}
    GEM1_PRO_50 : FB_ScrollPump;

(******************)
(******AT1L0*******)
(******************)
(*Gauges*)
    {attribute 'pytmc' :=' pv: AT1L0:GAS:GPI:10 '}
    {attribute 'TcLinkTo' := 	'.i_iPRESS_R	:=	TIIB[MKS_E7 (EL3064)]^AI Standard Channel 2^Value'}
    GATT_GPI_10 : FB_MKS317A;

    {attribute 'pytmc' :=' pv: AT1L0:GAS:GCM:11 '}
    {attribute 'TcLinkTo' := 	'.i_iPRESS_R	:=	TIIB[L0S6_PNL_04_EB_3 (EP4374-0002)]^AI Inputs Channel 1^Value'}
    GATT_GMP_11 : FB_CMR362;
    {attribute 'pytmc' :=' pv: AT1L0:GAS:GCM:10 '}
    {attribute 'TcLinkTo' := 	'.i_iPRESS_R	:=	TIIB[L0S6_PNL_04_EB_2 (EP3174-0002)]^AI Standard Channel 2^Value'}
    GATT_GMP_10 : FB_GCM;
(*Valves*)
    {attribute 'pytmc' :=' pv: AT1L0:GAS:VCN:10 '}
    GATT_VCN_10 : FB_VCN;
    {attribute 'pytmc' :=' pv: AT1L0:GAS:VRC:10 '}
    {attribute 'TcLinkTo' := 	'.i_xOpnLS	:=	TIIB[L0S6_PNL_04_EB_1 (EP2338-0002)]^Channel 1^Input;
                                 .i_xClsLS	:=	TIIB[L0S6_PNL_04_EB_1 (EP2338-0002)]^Channel 2^Input;
                                 .q_xOPN_DO	:=	TIIB[L0S6_PNL_04_EB_1 (EP2338-0002)]^Channel 11^Output'}
    GATT_VRC_10 : FB_VRC;

    {attribute 'pytmc' :=' pv: AT1L0:GAS:VVC:10 '}
    {attribute 'TcLinkTo' := 	'.q_xOPN_DO	:=	TIIB[L0S6_PNL_04_EB_1 (EP2338-0002)]^Channel 15^Output'}
    GATT_VVC_10: FB_VVC;



(******************)
(******EM2L0*******)
(******************)

(*Gauges*)
    {attribute 'pytmc' :=' pv: EM2L0:GEM:GPI:10 '}
    {attribute 'TcLinkTo' := 	'.i_iPRESS_R	:=	TIIB[MKS_E7 (EL3064)]^AI Standard Channel 4^Value'}
    GEM2_GPI_10 : FB_MKS317A;

    {attribute 'pytmc' :=' pv: EM2L0:GEM:GPI:11 '}
    {attribute 'TcLinkTo' := 	'.i_iPRESS_R	:=	TIIB[L0S6_PNL_01_EB_4 (EP3174-0002)]^AI Standard Channel 2^Value'}
    GEM2_GPI_11 : FB_MKS275;

    {attribute 'pytmc' :=' pv: EM2L0:GEM:GPI:21 '}
    {attribute 'TcLinkTo' := 	'.i_iPRESS_R	:=	TIIB[L0S6_PNL_01_EB_4 (EP3174-0002)]^AI Standard Channel 3^Value'}
    GEM2_GPI_21 : FB_MKS275;

    {attribute 'pytmc' :=' pv: EM2L0:GEM:GCC:30 '}
    {attribute 'TcLinkTo' := 	'.i_iPRESS_R	:=	TIIB[MKS_E7 (EL3064)]^AI Standard Channel 1^Value;
                                 .q_xHV_DIS		:= 	TIIB[MKS_E9 (EL2794)]^Channel 1^Output'}
    GEM2_GCC_30 : FB_MKS422;

    {attribute 'pytmc' :=' pv: EM2L0:GEM:GPI:30 '}
    {attribute 'TcLinkTo' := 	'.i_iPRESS_R	:=	TIIB[MKS_E7 (EL3064)]^AI Standard Channel 3^Value'}
    GEM2_GPI_30 : FB_MKS317A;

    {attribute 'pytmc' :=' pv: EM2L0:GEM:GPI:31 '}
    {attribute 'TcLinkTo' := 	'.i_iPRESS_R	:=	TIIB[L0S6_PNL_01_EB_4 (EP3174-0002)]^AI Standard Channel 4^Value'}
    GEM2_GPI_31 : FB_MKS275;

    {attribute 'pytmc' :=' pv: EM2L0:GEM:GCC:50 '}
    {attribute 'TcLinkTo' := 	'.i_iPRESS_R	:=	TIIB[MKS_E10 (EL3064)]^AI Standard Channel 1^Value;
                                 .q_xHV_DIS		:= 	TIIB[MKS_E12 (EL2794)]^Channel 1^Output'}
    GEM2_GCC_50 : FB_MKS422;

    {attribute 'pytmc' :=' pv: EM2L0:GEM:GPI:50 '}
    {attribute 'TcLinkTo' := 	'.i_iPRESS_R	:=	TIIB[MKS_E10 (EL3064)]^AI Standard Channel 4^Value'}
    GEM2_GPI_50 : FB_MKS317;

    {attribute 'pytmc' :=' pv: EM2L0:GEM:GPI:51 '}
    {attribute 'TcLinkTo' := 	'.i_iPRESS_R	:=	TIIB[L0S6_PNL_03_EB_6 (EP3174-0002)]^AI Standard Channel 2^Value'}
    GEM2_GPI_51 : FB_MKS275;

    {attribute 'pytmc' :=' pv: EM2L0:GEM:GCC:60 '}
    {attribute 'TcLinkTo' := 	'.i_iPRESS_R	:=	TIIB[MKS_E10 (EL3064)]^AI Standard Channel 3^Value;
                                 .q_xHV_DIS		:= 	TIIB[MKS_E12 (EL2794)]^Channel 2^Output'}
    GEM2_GCC_60 : FB_MKS422;
    {attribute 'pytmc' :=' pv: EM2L0:GEM:GPI:60 '}
    {attribute 'TcLinkTo' := 	'.i_iPRESS_R	:=	TIIB[MKS_E11 (EL3064)]^AI Standard Channel 1^Value'}
    GEM2_GPI_60 : FB_MKS317A;

    {attribute 'pytmc' :=' pv: EM2L0:GEM:GPI:61 '}
    {attribute 'TcLinkTo' := 	'.i_iPRESS_R	:=	TIIB[L0S6_PNL_03_EB_6 (EP3174-0002)]^AI Standard Channel 1^Value'}
    GEM2_GPI_61 : FB_MKS275;

    {attribute 'pytmc' :=' pv: EM2L0:GEM:GCC:70 '}
    {attribute 'TcLinkTo' := 	'.i_iPRESS_R	:=	TIIB[MKS_E13 (EL3064)]^AI Standard Channel 1^Value;
                                 .q_xHV_DIS		:= 	TIIB[MKS_E15 (EL2794)]^Channel 1^Output'}
    GEM2_GCC_70 : FB_MKS422;

    {attribute 'pytmc' :=' pv: EM2L0:GEM:GPI:70 '}
    {attribute 'TcLinkTo' := 	'.i_iPRESS_R	:=	TIIB[MKS_E13 (EL3064)]^AI Standard Channel 4^Value'}
    GEM2_GPI_70 : FB_MKS317A;

(* GAS Cell CM*)

    {attribute 'pytmc' :=' pv: EM2L0:GEM:GCM:41 '}
    {attribute 'TcLinkTo' := 	'.i_iPRESS_R	:=	TIIB[L0S6_PNL_02_EB_4 (EP3174-0002)]^AI Standard Channel 1^Value'}
    GEM2_GCM_41 : FB_GCM;
    {attribute 'pytmc' :=' pv: EM2L0:GEM:GCM:42 '}
    {attribute 'TcLinkTo' := 	'.i_iPRESS_R	:=	TIIB[L0S6_PNL_02_EB_4 (EP3174-0002)]^AI Standard Channel 2^Value'}
    GEM2_GCM_42 : FB_GCM;
    (*Pseudo gauge device Structure to combine the readings of two GCM gauges*)
    {attribute 'pytmc' :=' pv: EM2L0:GEM:GCM:40 '}
    GEM2_GCM_40 : ST_VG;

(*valves*)

    {attribute 'pytmc' :=' pv: EM2L0:GEM:VGC:10 '}
    {attribute 'TcLinkTo' := 	'.i_xOpnLS	:=	TIIB[L0S6_PNL_01_EB_1 (EP2338-0002)]^Channel 1^Input;
                                 .i_xClsLS	:=	TIIB[L0S6_PNL_01_EB_1 (EP2338-0002)]^Channel 2^Input;
                                 .q_xOPN_DO	:=	TIIB[L0S6_PNL_01_EB_1 (EP2338-0002)]^Channel 11^Output'}
    GEM2_VGC_10: FB_VGC;

    {attribute 'pytmc' :=' pv: EM2L0:GEM:VGC:20'}
    {attribute 'TcLinkTo' := 	'.i_xOpnLS	:=	TIIB[L0S6_PNL_01_EB_1 (EP2338-0002)]^Channel 5^Input;
                                 .i_xClsLS	:=	TIIB[L0S6_PNL_01_EB_1 (EP2338-0002)]^Channel 6^Input;
                                 .q_xOPN_DO	:=	TIIB[L0S6_PNL_01_EB_1 (EP2338-0002)]^Channel 15^Output'}
    GEM2_VGC_20: FB_VGC;

    {attribute 'pytmc' :=' pv: EM2L0:GEM:VGC:30 '}
    {attribute 'TcLinkTo' := 	'.i_xOpnLS	:=	TIIB[L0S6_PNL_02_EB_1 (EP2338-0002)]^Channel 1^Input;
                                 .i_xClsLS	:=	TIIB[L0S6_PNL_02_EB_1 (EP2338-0002)]^Channel 2^Input;
                                 .q_xOPN_DO	:=	TIIB[L0S6_PNL_02_EB_1 (EP2338-0002)]^Channel 11^Output'}
    GEM2_VGC_30: FB_VGC;

    {attribute 'pytmc' :=' pv: EM2L0:GEM:VGC:40 '}
    {attribute 'TcLinkTo' := 	'.i_xOpnLS	:=	TIIB[L0S6_PNL_02_EB_1 (EP2338-0002)]^Channel 5^Input;
                                 .i_xClsLS	:=	TIIB[L0S6_PNL_02_EB_1 (EP2338-0002)]^Channel 6^Input;
                                 .q_xOPN_DO	:=	TIIB[L0S6_PNL_02_EB_1 (EP2338-0002)]^Channel 15^Output'}
    GEM2_VGC_40: FB_VGC;

    {attribute 'pytmc' :=' pv: EM2L0:GEM:VGC:50 '}
    {attribute 'TcLinkTo' := 	'.i_xOpnLS	:=	TIIB[L0S6_PNL_03_EB_1 (EP2338-0002)]^Channel 1^Input;
                                 .i_xClsLS	:=	TIIB[L0S6_PNL_03_EB_1 (EP2338-0002)]^Channel 2^Input;
                                 .q_xOPN_DO	:=	TIIB[L0S6_PNL_03_EB_1 (EP2338-0002)]^Channel 11^Output'}
    GEM2_VGC_50: FB_VGC;

    {attribute 'pytmc' :=' pv: EM2L0:GEM:VGC:60 '}
    {attribute 'TcLinkTo' := 	'.i_xOpnLS	:=	TIIB[L0S6_PNL_03_EB_3 (EP2338-0002)]^Channel 1^Input;
                                 .i_xClsLS	:=	TIIB[L0S6_PNL_03_EB_3 (EP2338-0002)]^Channel 2^Input;
                                 .q_xOPN_DO	:=	TIIB[L0S6_PNL_03_EB_3 (EP2338-0002)]^Channel 11^Output'}
    GEM2_VGC_60: FB_VGC;

    {attribute 'pytmc' :=' pv: EM2L0:GEM:VGC:70 '}
    {attribute 'TcLinkTo' := 	'.i_xOpnLS	:=	TIIB[L0S6_PNL_03_EB_3 (EP2338-0002)]^Channel 5^Input;
                                 .i_xClsLS	:=	TIIB[L0S6_PNL_03_EB_3 (EP2338-0002)]^Channel 6^Input;
                                 .q_xOPN_DO	:=	TIIB[L0S6_PNL_03_EB_3 (EP2338-0002)]^Channel 15^Output'}
    GEM2_VGC_70: FB_VGC;

(*Turbo isolation valves*)

    {attribute 'pytmc' :=' pv: EM2L0:GEM:VRC:30 '}
    {attribute 'TcLinkTo' := 	'.i_xOpnLS	:=	TIIB[L0S6_PNL_01_EB_3 (EP2338-0002)]^Channel 1^Input;
                                 .i_xClsLS	:=	TIIB[L0S6_PNL_01_EB_3 (EP2338-0002)]^Channel 2^Input;
                                 .q_xOPN_DO	:=	TIIB[L0S6_PNL_01_EB_3 (EP2338-0002)]^Channel 11^Output'}
    GEM2_VRC_30: FB_VRC;
    {attribute 'pytmc' :=' pv: EM2L0:GEM:VRC:50 '}
    {attribute 'TcLinkTo' := 	'.i_xOpnLS	:=	TIIB[L0S6_PNL_03_EB_1 (EP2338-0002)]^Channel 5^Input;
                                 .i_xClsLS	:=	TIIB[L0S6_PNL_03_EB_1 (EP2338-0002)]^Channel 6^Input;
                                 .q_xOPN_DO	:=	TIIB[L0S6_PNL_03_EB_1 (EP2338-0002)]^Channel 15^Output'}
    GEM2_VRC_50: FB_VRC;

    {attribute 'pytmc' :=' pv: EM2L0:GEM:VRC:60 '}
    {attribute 'TcLinkTo' := 	'.i_xOpnLS	:=	TIIB[L0S6_PNL_03_EB_2 (EP2338-0002)]^Channel 1^Input;
                                 .i_xClsLS	:=	TIIB[L0S6_PNL_03_EB_2 (EP2338-0002)]^Channel 2^Input;
                                 .q_xOPN_DO	:=	TIIB[L0S6_PNL_03_EB_2 (EP2338-0002)]^Channel 11^Output'}
    GEM2_VRC_60: FB_VRC;

    {attribute 'pytmc' :=' pv: EM2L0:GEM:VRC:70 '}
    {attribute 'TcLinkTo' := 	'.i_xOpnLS	:=	TIIB[L0S6_PNL_03_EB_2 (EP2338-0002)]^Channel 5^Input;
                                 .i_xClsLS	:=	TIIB[L0S6_PNL_03_EB_2 (EP2338-0002)]^Channel 6^Input;
                                 .q_xOPN_DO	:=	TIIB[L0S6_PNL_03_EB_2 (EP2338-0002)]^Channel 15^Output'}
    GEM2_VRC_70: FB_VRC;

(*Kashiyama*)
    {attribute 'pytmc' :=' pv: EM2L0:GEM:VRC:10 '}
    {attribute 'TcLinkTo' := 	'.i_xOpnLS	:=	TIIB[L0S6_PNL_01_EB_2 (EP2338-0002)]^Channel 1^Input;
                                 .i_xClsLS	:=	TIIB[L0S6_PNL_01_EB_2 (EP2338-0002)]^Channel 2^Input;
                                 .q_xOPN_DO	:=	TIIB[L0S6_PNL_01_EB_2 (EP2338-0002)]^Channel 11^Output'}
    GEM2_VRC_10:FB_Kashiyama_VRC;

    {attribute 'pytmc' :=' pv: EM2L0:GEM:VRC:20 '}
    {attribute 'TcLinkTo' := 	'.i_xOpnLS	:=	TIIB[L0S6_PNL_01_EB_2 (EP2338-0002)]^Channel 5^Input;
                                 .i_xClsLS	:=	TIIB[L0S6_PNL_01_EB_2 (EP2338-0002)]^Channel 6^Input;
                                 .q_xOPN_DO	:=	TIIB[L0S6_PNL_01_EB_2 (EP2338-0002)]^Channel 15^Output'}
    GEM2_VRC_20:FB_Kashiyama_VRC;

(*Turbo vent valves*) (*deprecated*)
    {attribute 'pytmc' :=' pv: EM2L0:GEM:VVC:30 '}
    {attribute 'TcLinkTo' := 	'.q_xCLS_DO	:=	TIIB[L0S6_PNL_01_EB_3 (EP2338-0002)]^Channel 15^Output'}
    GEM2_VVC_30: FB_TurbVentvalve_NO;
    {attribute 'pytmc' :=' pv: EM2L0:GEM:VVC:50 '}
    {attribute 'TcLinkTo' := 	'.q_xCLS_DO	:=	TIIB[L0S6_PNL_03_EB_4 (EP2338-0002)]^Channel 15^Output'}
    GEM2_VVC_50: FB_TurbVentvalve_NO;
    {attribute 'pytmc' :=' pv: EM2L0:GEM:VVC:70 '}
    {attribute 'TcLinkTo' := 	'.q_xCLS_DO	:=	TIIB[L0S6_PNL_03_EB_4 (EP2338-0002)]^Channel 16^Output'}
    GEM2_VVC_70: FB_TurbVentvalve_NO;

(*Gas cell vent valve*)
    {attribute 'pytmc' :=' pv: EM2L0:GEM:VVC:40 '}
    {attribute 'TcLinkTo' := 	'.q_xOPN_DO	:=	TIIB[L0S6_PNL_02_EB_2 (EP2338-0002)]^Channel 15^Output'}
    GEM2_VVC_40: FB_VVC;
(*Pressure Control Valve*)
    {attribute 'pytmc' :=' pv: EM2L0:GEM:VCN:40 '}
    {attribute 'TcLinkTo' := 	'.q_iRawPosition	:=	TIIB[L0S6_PNL_02_EB_3 (EP4374-0002)]^AO Outputs Channel 4^Analog output'}
    GEM2_VCN_40 : FB_VCN;


(*Pumps*)
(*Turbos*)
(*REMOVE
    {attribute 'pytmc' :=' pv: EM2L0:GEM:PTM:30 '}
    {attribute 'TcLinkTo' := 	'.i_xR1	:=	TIIB[PLC_EL_7 (EL1088)]^Channel 1^Input;
                                 .i_xLSpd :=	TIIB[PLC_EL_7 (EL1088)]^Channel 2^Input;
                                 .i_xSTART	:=	TIIB[PLC_EL_7 (EL1088)]^Channel 3^Input;
                                 .i_xFault	:=	TIIB[PLC_EL_7 (EL1088)]^Channel 4^Input;
                                 .i_iCurrentMon := TIIB[PLC_EL_5 (EL3064)]^AI Standard Channel 1^Value;
                                 .q_RunDO	:=	TIIB[PLC_EL_6 (EL2088)]^Channel 1^Output'}
    GEM2_PTM_30 : FB_PTM_Agilent;
    *)
    {attribute 'pytmc' :=' pv: EM2L0:GEM:PTM:30 '}
    {attribute 'TcLinkTo' := 	'.i_xDecel	:=	TIIB[PTM_E11_EL1004]^Channel 1^Input;
                                 .i_xAtSpd	:=	TIIB[PTM_E11_EL1004]^Channel 2^Input;
                                 .i_xNCFault :=	TIIB[PTM_E11_EL1004]^Channel 3^Input;
                                 .i_xRotate	:=	TIIB[PTM_E11_EL1004]^Channel 4^Input;
                                 .i_xAccel :=	TIIB[PTM_E12_EL1004]^Channel 1^Input;
                                 .i_iRawSpeed := TIIB[PTM_E14_EL3064]^AI Standard Channel 1^Value;
                                 .i_iCurrentMon := TIIB[PTM_E14_EL3064]^AI Standard Channel 2^Value;
                                 .i_iTempMon := TIIB[PTM_E14_EL3064]^AI Standard Channel 3^Value;
                                 .q_xReset	:=	TIIB[PTM_E13_EL2798]^Channel 1^Output;
                                 .q_xStart	:=	TIIB[PTM_E13_EL2798]^Channel 2^Output;
                                 .q_xStop	:=	TIIB[PTM_E13_EL2798]^Channel 3^Output;
                                 .q_xProtection	:=	TIIB[PTM_E13_EL2798]^Channel 4^Output;
                                 .q_xSetSpeed	:=	TIIB[PTM_E13_EL2798]^Channel 5^Output;
                                 .q_iSpeedSet	:=	TIIB[PTM_E15_EL4004]^AO Outputs Channel 1^Analog output'}
    GEM2_PTM_30 : FB_PTM_Ebara_010M;
    (*REMOVE{attribute 'pytmc' :=' pv: EM2L0:GEM:PTM:50 '}
    {attribute 'TcLinkTo' := 	'.i_xR1	:=	TIIB[PLC_EL_7 (EL1088)]^Channel 5^Input;
                                 .i_xLSpd :=	TIIB[PLC_EL_7 (EL1088)]^Channel 6^Input;
                                 .i_xSTART	:=	TIIB[PLC_EL_7 (EL1088)]^Channel 7^Input;
                                 .i_xFault	:=	TIIB[PLC_EL_7 (EL1088)]^Channel 8^Input;
                                 .i_iCurrentMon := TIIB[PLC_EL_5 (EL3064)]^AI Standard Channel 2^Value;
                                 .q_RunDO	:=	TIIB[PLC_EL_6 (EL2088)]^Channel 2^Output'}
    GEM2_PTM_50 : FB_PTM_Agilent;*)

    {attribute 'pytmc' :=' pv: EM2L0:GEM:PTM:50 '}
    {attribute 'TcLinkTo' := 	'.i_xDecel	:=	TIIB[PTM_E18_EL1004]^Channel 1^Input;
                                 .i_xAtSpd	:=	TIIB[PTM_E18_EL1004]^Channel 2^Input;
                                 .i_xNCFault :=	TIIB[PTM_E18_EL1004]^Channel 3^Input;
                                 .i_xRotate	:=	TIIB[PTM_E18_EL1004]^Channel 4^Input;
                                 .i_xAccel :=	TIIB[PTM_E19_EL1004]^Channel 1^Input;
                                 .i_iRawSpeed := TIIB[PTM_E16_EL3064]^AI Standard Channel 1^Value;
                                 .i_iCurrentMon := TIIB[PTM_E16_EL3064]^AI Standard Channel 2^Value;
                                 .i_iTempMon := TIIB[PTM_E16_EL3064]^AI Standard Channel 3^Value;
                                 .q_xReset	:=	TIIB[PTM_E17_EL2798]^Channel 1^Output;
                                 .q_xStart	:=	TIIB[PTM_E17_EL2798]^Channel 2^Output;
                                 .q_xStop	:=	TIIB[PTM_E17_EL2798]^Channel 3^Output;
                                 .q_xProtection	:=	TIIB[PTM_E17_EL2798]^Channel 4^Output;
                                 .q_xSetSpeed	:=	TIIB[PTM_E17_EL2798]^Channel 5^Output;
                                 .q_iSpeedSet	:=	TIIB[PTM_E15_EL4004]^AO Outputs Channel 3^Analog output'}
    GEM2_PTM_50 : FB_PTM_Ebara_010M;
    (*REMOVE{attribute 'pytmc' :=' pv: EM2L0:GEM:PTM:60 '}
    {attribute 'TcLinkTo' := 	'.i_xR1	:=	TIIB[PLC_EL_8 (EL1088)]^Channel 1^Input;
                                 .i_xLSpd :=	TIIB[PLC_EL_8 (EL1088)]^Channel 2^Input;
                                 .i_xSTART	:=	TIIB[PLC_EL_8 (EL1088)]^Channel 3^Input;
                                 .i_xFault	:=	TIIB[PLC_EL_8 (EL1088)]^Channel 4^Input;
                                 .i_iPowerMon := TIIB[PLC_EL_5 (EL3064)]^AI Standard Channel 3^Value;
                                 .q_RunDO	:=	TIIB[PLC_EL_6 (EL2088)]^Channel 3^Output'}
    GEM2_PTM_60 : FB_PTM_Agilent;
    *)
    {attribute 'pytmc' :=' pv: EM2L0:GEM:PTM:60 '}
    {attribute 'TcLinkTo' := 	'.i_xAtSpd	:=	TIIB[PTM_E21_EL1088]^Channel 5^Input;
                                 .i_xFault :=	TIIB[PTM_E21_EL1088]^Channel 6^Input;
                                 .q_RunDO	:=	TIIB[PTM_E20_EL2624]^Channel 3^Output'}
    GEM2_PTM_60 : FB_PTM_TwisTorr;
    {attribute 'pytmc' :=' pv: EM2L0:GEM:PTM:70 '}
    {attribute 'TcLinkTo' := 	'.i_xAtSpd	:=	TIIB[PTM_E21_EL1088]^Channel 7^Input;
                                 .i_xFault :=	TIIB[PTM_E21_EL1088]^Channel 8^Input;
                                 .q_RunDO	:=	TIIB[PTM_E20_EL2624]^Channel 4^Output'}
    GEM2_PTM_70 : FB_PTM_TwisTorr;//FB_PTM_Agilent;




(*Scroll Pumps*)
    {attribute 'pytmc' :=' pv: EM2L0:GEM:PRO:30 '}
    {attribute 'TcLinkTo' := 	'.q_xRunDo	:=	TIIB[L0S6_PNL_01_EB_7 (EP2338-0002)]^Channel 11^Output'}
    GEM2_PRO_30 : FB_ScrollPump;
    {attribute 'pytmc' :=' pv: EM2L0:GEM:PRO:50 '}
    {attribute 'TcLinkTo' := 	'.q_xRunDo	:=	TIIB[L0S6_PNL_01_EB_7 (EP2338-0002)]^Channel 12^Output'}
    GEM2_PRO_50 : FB_ScrollPump;
    {attribute 'pytmc' :=' pv: EM2L0:GEM:PRO:60 '}
    {attribute 'TcLinkTo' := 	'.q_xRunDo	:=	TIIB[L0S6_PNL_01_EB_7 (EP2338-0002)]^Channel 15^Output'}
    GEM2_PRO_60 : FB_ScrollPump;
(*Kashyiama Dry Pumps*)

    {attribute 'pytmc' :=' pv: EM2L0:GEM:PRO:10 '}
    {attribute 'TcLinkTo' := 	'.i_xIsRun	:=	TIIB[L0S6_PNL_01_EB_7 (EP2338-0002)]^Channel 1^Input;
                                 .i_xLocal	:=	TIIB[L0S6_PNL_01_EB_7 (EP2338-0002)]^Channel 2^Input;
                                 .i_xWarning :=	TIIB[L0S6_PNL_01_EB_7 (EP2338-0002)]^Channel 5^Input;
                                 .i_xAlarm :=	TIIB[L0S6_PNL_01_EB_7 (EP2338-0002)]^Channel 6^Input;
                                 .q_xRunDO	:=	TIIB[L0S6_PNL_01_EB_6 (EP2624-0002)]^Channel 1^Output;
                                 .q_xLspdDo	:=	TIIB[L0S6_PNL_01_EB_6 (EP2624-0002)]^Channel 2^Output;
                                 .q_xResetDo:=	TIIB[L0S6_PNL_01_EB_6 (EP2624-0002)]^Channel 3^Output'}
    GEM2_PRO_10: FB_KashiyamaPump;
    {attribute 'pytmc' :=' pv: EM2L0:GEM:PRO:20 '}
    {attribute 'TcLinkTo' := 	'.i_xIsRun	:=	TIIB[L0S6_PNL_01_EB_9 (EP2338-0002)]^Channel 1^Input;
                                 .i_xLocal	:=	TIIB[L0S6_PNL_01_EB_9 (EP2338-0002)]^Channel 2^Input;
                                 .i_xWarning :=	TIIB[L0S6_PNL_01_EB_9 (EP2338-0002)]^Channel 5^Input;
                                 .i_xAlarm :=	TIIB[L0S6_PNL_01_EB_9 (EP2338-0002)]^Channel 6^Input;
                                 .q_xRunDO	:=	TIIB[L0S6_PNL_01_EB_8 (EP2624-0002)]^Channel 1^Output;
                                 .q_xLspdDo	:=	TIIB[L0S6_PNL_01_EB_8 (EP2624-0002)]^Channel 2^Output;
                                 .q_xResetDo:=	TIIB[L0S6_PNL_01_EB_8 (EP2624-0002)]^Channel 3^Output'}
    GEM2_PRO_20: FB_KashiyamaPump;


END_VAR

// ---- GVLs/GVL_ILK.TcGVL
VAR_GLOBAL

    {attribute 'pytmc' := '
    pv: PLC:LFE:GEM:FFO:01
    '}
    {attribute 'TcLinkTo' := '.q_xFastFaultOut:=TIIB[PMPS_FFO]^Channel 1^Output'}
    g_FastFaultOutput1  :   FB_HardwareFFOutput :=(i_sNetID:='172.21.88.66.1.1');

    {attribute 'pytmc' := '
    pv: PLC:LFE:GEM:FFO:02
    '}
    {attribute 'TcLinkTo' := '.q_xFastFaultOut:=TIIB[PMPS_FFO]^Channel 2^Output'}
    g_FastFaultOutput2  :   FB_HardwareFFOutput :=(i_sNetID:='172.21.88.66.1.1');

    {attribute 'pytmc' := 'pv: EM1L0:GEM:ARB:01'}
    g_fbArbiter   :   FB_Arbiter(1);
    {attribute 'pytmc' := 'pv: EM1L0:GEM:ARB:02'}
    g_fbArbiter2   :   FB_Arbiter(2);
    {attribute 'pytmc' := 'pv: EM1L0:GEM:ARB:03'}
    g_fbArbiter3   :   FB_Arbiter(3);



    {attribute 'pytmc' := 'pv: EM1L0:GEM:VAC:OVRDON;
    field: ZNAM Override OFF;
    field: ONAM Override ON;
     io: io;
    '}
    xGEM1OverrideMode	:	BOOL; (* Global system override for the EM1L0*)
    {attribute 'pytmc' := 'pv: AT1L0:GAS:VAC:OVRDON;
    field: ZNAM Override OFF;
    field: ONAM Override ON;
     io: io;
    '}
    xGATTOverrideMode	:	BOOL; (* Global system override for the GATT*)
    {attribute 'pytmc' := 'pv: EM2L0:GEM:VAC:OVRDON;
    field: ZNAM Override OFF;
    field: ONAM Override ON;
     io: io;
    '}
    xGEM2OverrideMode	:	BOOL; (* Global system override for the EM2L0*)


(* Interlock related bits, local to the PLC*)
    GEM1_Turbo_Valves_Closed:  BOOL;
    GEM1_Turbo_Valves_Open:  BOOL;
    GEM2_Turbo_Valves_Closed: BOOL;
    GEM2_Turbo_Valves_Open:  BOOL;
    GEM1_Turbo_Running:  BOOL;
    GEM2_Turbo_Running:  BOOL;
    TwinscrewPumps_Valves_Closed: BOOL;
    GEM1_TwinscrewPumps_Valves_Open : BOOL;
    GEM2_TwinscrewPumps_Valves_Open : BOOL;
    GEM1_Aperture_Closed: BOOL;
    GEM2_Aperture_Closed: BOOL;

    xGEM1_AperturesOpnOK : BOOL;
    xGEM2_AperturesOpnOK : BOOL;



END_VAR

// ---- GVLs/GVL_Sensors.TcGVL
VAR_GLOBAL

(*Pressure Meter*)
    {attribute 'pytmc' :=' pv: EM1L0:GEM:AIR:1 '}
    GEM1_AIR_1 :FB_PressureSensor_PX219;
    {attribute 'pytmc' :=' pv: EM1L0:GEM:AIR:2 '}
    GEM1_AIR_2 :FB_PressureSensor_PX219;
    {attribute 'pytmc' :=' pv: EM2L0:GEM:N2:1 '}
    GEM2_N2_1 :FB_PressureSensor_PX219;
    {attribute 'pytmc' :=' pv: EM2L0:GEM:N2:2 '}
    GEM2_N2_2 :FB_PressureSensor_PX219;
    (*Flow Meters*)
    {attribute 'pytmc' :=' pv: EM1L0:GEM:GFM:41 '}
    GEM1_GFM_41 :FB_PressureSensor_PX219;
    {attribute 'pytmc' :=' pv: EM1L0:GEM:GFM:42 '}
    GEM1_GFM_42 :FB_PressureSensor_PX219;
    {attribute 'pytmc' :=' pv: EM2L0:GEM:GFM:41 '}
    GEM2_GFM_41 :FB_PressureSensor_PX219;
    {attribute 'pytmc' :=' pv: EM2L0:GEM:GFM:42 '}
    GEM2_GFM_42 :FB_PressureSensor_PX219;

END_VAR

// ---- POUs/MAIN.TcPOU
PROGRAM MAIN
VAR
    iWatchdog:UDINT;//The watchdog variable name written to by the remote plc

    fbLogHandler: FB_LogHandler;
END_VAR

(*Ethercat Diagnostics*)
//DIAGNOSTICS();



(* Call all Programs*)
PRG_ILK();
PRG_GEM1_DIFF_PUMP();
PRG_GEM2_DIFF_PUMP();
PRG_ROOTS();
PRG_GATT();
PRG_GEM1();
PRG_GEM2();
PRG_PMPS();
//Log Handler
fbLogHandler();

END_PROGRAM

// ---- POUs/PRG_ILK.TcPOU
PROGRAM PRG_ILK
VAR
END_VAR

(*Evaluate Global Interlocks*)

TwinscrewPumps_Valves_Closed := GEM1_VRC_60.q_stValve.i_xClsLS AND  GEM1_VRC_70.q_stValve.i_xClsLS AND GEM2_VRC_10.q_stValve.i_xClsLS AND GEM2_VRC_20.q_stValve.i_xClsLS;
GEM1_Turbo_Valves_Closed := GEM1_VRC_10.iq_stValve.i_xClsLS AND  GEM1_VRC_20.iq_stValve.i_xClsLS AND GEM1_VRC_30.iq_stValve.i_xClsLS AND GEM1_VRC_50.iq_stValve.i_xClsLS;
GEM2_Turbo_Valves_Closed := GEM2_VRC_30.iq_stValve.i_xClsLS AND  GEM2_VRC_50.iq_stValve.i_xClsLS AND GEM2_VRC_60.iq_stValve.i_xClsLS AND GEM2_VRC_70.iq_stValve.i_xClsLS;
GEM1_TwinscrewPumps_Valves_Open := (GEM1_VRC_60.q_stValve.i_xOpnLS AND GEM1_PRO_60.q_stPump.i_xIsRun) OR   (GEM1_VRC_70.q_stValve.i_xOpnLS AND GEM1_PRO_70.q_stPump.i_xIsRun);
GEM2_TwinscrewPumps_Valves_Open := (GEM2_VRC_10.q_stValve.i_xOpnLS AND GEM2_PRO_10.q_stPump.i_xIsRun) OR   (GEM2_VRC_20.q_stValve.i_xOpnLS AND GEM2_PRO_20.q_stPump.i_xIsRun);
GEM1_Turbo_Valves_Open := GEM1_VRC_10.iq_stValve.i_xOpnLS AND  GEM1_VRC_20.iq_stValve.i_xOpnLS AND GEM1_VRC_30.iq_stValve.i_xOpnLS AND GEM1_VRC_50.iq_stValve.i_xOpnLS;
GEM2_Turbo_Valves_Open := GEM2_VRC_30.iq_stValve.i_xOpnLS AND  GEM2_VRC_50.iq_stValve.i_xOpnLS AND GEM2_VRC_60.iq_stValve.i_xOpnLS AND GEM2_VRC_70.iq_stValve.i_xOpnLS; (*MG 03.09.20 Turbo is failing, but injection can run without it*)
GEM1_Aperture_Closed :=  GEM1_VGC_20.iq_stValve.i_xClsLS AND GEM1_VGC_30.iq_stValve.i_xClsLS AND GEM1_VGC_40.iq_stValve.i_xClsLS AND GEM1_VGC_50.iq_stValve.i_xClsLS AND GEM1_VGC_60.iq_stValve.i_xClsLS AND GEM1_VGC_70.iq_stValve.i_xClsLS ;
GEM2_Aperture_Closed := GEM2_VGC_10.iq_stValve.i_xClsLS AND GEM2_VGC_20.iq_stValve.i_xClsLS AND GEM2_VGC_30.iq_stValve.i_xClsLS AND GEM2_VGC_40.iq_stValve.i_xClsLS AND GEM2_VGC_50.iq_stValve.i_xClsLS AND GEM2_VGC_60.iq_stValve.i_xClsLS; ;
GEM1_Turbo_Running := (GEM1_PTM_10.iq_stPtm.eState = pumpRUNNING) AND (GEM1_PTM_20.iq_stPtm.eState = pumpRUNNING) AND (GEM1_PTM_30.iq_stPtm.eState = pumpRUNNING) AND (GEM1_PTM_50.iq_stPtm.eState = pumpRUNNING);
GEM2_Turbo_Running := (GEM2_PTM_30.iq_stPtm.eState = pumpRUNNING) AND (GEM2_PTM_50.iq_stPtm.eState = pumpRUNNING) AND (GEM2_PTM_60.iq_stPtm.eState = pumpRUNNING) AND (GEM2_PTM_70.iq_stPtm.eState = pumpRUNNING); (*MG 03.09.20 Turbo is failing, but injection can run without it*)

xGEM1_AperturesOpnOK := NOT GEM1_VVC_40.iq_stValve.q_xOPN_DO AND NOT GATT_VVC_10.iq_stValve.q_xOPN_DO; //AND VCN is closed
xGEM2_AperturesOpnOK := NOT GEM2_VVC_40.iq_stValve.q_xOPN_DO AND NOT GATT_VVC_10.iq_stValve.q_xOPN_DO; //AND VCN is closed

(* Link The correct override bit to the correct vacuum section*)



(*P/MPS FF*)

END_PROGRAM

// ---- POUs/PRG_GEM1_DIFF_PUMP.TcPOU
PROGRAM PRG_GEM1_DIFF_PUMP
VAR
    rMaxBackingPressure : REAL := 0.7;//Torr
    bInit:BOOL:=TRUE;

END_VAR

If (bInit) THEN
    bInit := FALSE;
    //GEM1_PTM_10.M_SetPowerScale(15);
    //GEM1_PTM_20.M_SetPowerScale(15);
END_IF

(*Gauges*)
USG_PIN(sNetId:='172.21.88.138.1.1' , nPort:=851 , sVarName:='GVL_Devices.SL1L0_POWER_PIN_01',iWatchdog:=Main.iWatchdog,IG=> );
USG_GCC(sNetId:='172.21.88.138.1.1' , nPort:=851 , sVarName:='GVL_Devices.SL1L0_POWER_GCC_01',iWatchdog:=Main.iWatchdog,IG=> );

GEM1_GPI_10(PG=>);
GEM1_GCC_10(PG:=GEM1_GPI_10.PG,IG=>);
GEM1_GPI_20(PG=>);
GEM1_GCC_20(PG:=GEM1_GPI_20.PG,IG=>);
GEM1_GPI_30(PG=>);
GEM1_GCC_30(PG:=GEM1_GPI_30.PG,IG=>);
GEM1_GPI_50(PG=>);
GEM1_GCC_50(PG:=GEM1_GPI_50.PG,IG=>);
GEM1_GPI_11(PG=>);
GEM1_GPI_31(PG=>);
GEM1_GPI_51(PG=>);

(*VALVES*)
(*Aperture valve may open when Detector and Attenuator N2 valves are closed. Override provided *)
 (* to Include PMPS ILK with the EXTILK bit*)
(*apperture valves*)

GEM1_VGC_10(i_stUSG := USG_GCC.IG, i_stDSG:= GEM1_GCC_10.IG,i_xDis_DPIlk := FALSE, i_xEPS_OK := TRUE,
        i_xPMPS_OK := TRUE, i_xExt_OK := NOT (USG_GCC.bError), i_xOverrideMode := xGEM1OverrideMode,i_xReset := ,
        io_fbFFHWO :=g_FastFaultOutput1,i_sDevName:= 'EM1L0:GEM:VGC:10',fbArbiter:=g_fbArbiter,i_nTransitionRootID:=1100);
GEM1_VGC_20(i_stUSG := GEM1_GCC_10.IG, i_stDSG:= GEM1_GCC_20.IG,i_xDis_DPIlk := TRUE, i_xEPS_OK := TRUE,
        i_xPMPS_OK := TRUE, i_xExt_OK := xGEM1_AperturesOpnOK, i_xOverrideMode := xGEM1OverrideMode,i_xReset := , i_xIsAperture:= TRUE ,
        io_fbFFHWO :=g_FastFaultOutput1,i_sDevName:= 'EM1L0:GEM:VGC:20',fbArbiter:=g_fbArbiter,i_nTransitionRootID:=1200);
GEM1_VGC_30(i_stUSG := GEM1_GCC_20.IG, i_stDSG:= GEM1_GCC_30.IG,i_xDis_DPIlk := TRUE, i_xEPS_OK := TRUE,
        i_xPMPS_OK := TRUE, i_xExt_OK := xGEM1_AperturesOpnOK, i_xOverrideMode := xGEM1OverrideMode,i_xReset := , i_xIsAperture:= TRUE ,
        io_fbFFHWO :=g_FastFaultOutput1,i_sDevName:= 'EM1L0:GEM:VGC:30',fbArbiter:=g_fbArbiter,i_nTransitionRootID:=1300);
GEM1_VGC_40(i_stUSG := GEM1_GCC_30.IG, i_stDSG:= GEM1_GCC_30.IG,i_xDis_DPIlk := TRUE, i_xEPS_OK := TRUE,
        i_xPMPS_OK := TRUE, i_xExt_OK := xGEM1_AperturesOpnOK, i_xOverrideMode := xGEM1OverrideMode,i_xReset := , i_xIsAperture:= TRUE,
        io_fbFFHWO :=g_FastFaultOutput1,i_sDevName:= 'EM1L0:GEM:VGC:40',fbArbiter:=g_fbArbiter,i_nTransitionRootID:=1400);
GEM1_VGC_50(i_stUSG := GEM1_GCC_50.IG, i_stDSG:= GEM1_GCC_50.IG,i_xDis_DPIlk := TRUE, i_xEPS_OK := TRUE,
        i_xPMPS_OK := TRUE, i_xExt_OK := xGEM1_AperturesOpnOK, i_xOverrideMode := xGEM1OverrideMode,i_xReset := , i_xIsAperture:= TRUE ,
        io_fbFFHWO :=g_FastFaultOutput1,i_sDevName:= 'EM1L0:GEM:VGC:50',fbArbiter:=g_fbArbiter,i_nTransitionRootID:=1500);
GEM1_VGC_60(i_stUSG := GEM1_GCC_50.IG, i_stDSG:= GEM1_GCC_50.IG,i_xDis_DPIlk := TRUE, i_xEPS_OK := TRUE,
        i_xPMPS_OK := TRUE, i_xExt_OK := xGEM1_AperturesOpnOK, i_xOverrideMode := xGEM1OverrideMode,i_xReset := , i_xIsAperture:= TRUE ,
        io_fbFFHWO :=g_FastFaultOutput1,i_sDevName:= 'EM1L0:GEM:VGC:60',fbArbiter:=g_fbArbiter,i_nTransitionRootID:=1600);
GEM1_VGC_70(i_stUSG := GEM1_GCC_50.IG, i_stDSG:= GEM1_GCC_50.IG,i_xDis_DPIlk := TRUE, i_xEPS_OK := TRUE,
        i_xPMPS_OK := TRUE, i_xExt_OK := xGEM1_AperturesOpnOK, i_xOverrideMode := xGEM1OverrideMode,i_xReset := , i_xIsAperture:= TRUE ,
        io_fbFFHWO:=g_FastFaultOutput1,i_sDevName:= 'EM1L0:GEM:VGC:70',fbArbiter:=g_fbArbiter,i_nTransitionRootID:=1700);

(*Turbo Isolation Valves*)
 GEM1_VRC_10(i_xExtILK_OK := F_TurboGateValve_ILK(GEM1_PTM_10.iq_stPtm,GEM1_GPI_10.PG) AND GEM1_PTM_10.iq_stPtm.eState = pumpRUNNING ,i_xOverrideMode := xGEM1OverrideMode);
 GEM1_VRC_20(i_xExtILK_OK := F_TurboGateValve_ILK(GEM1_PTM_20.iq_stPtm,GEM1_GPI_20.PG) AND GEM1_PTM_20.iq_stPtm.eState = pumpRUNNING,i_xOverrideMode := xGEM1OverrideMode);
 GEM1_VRC_30(i_xExtILK_OK := F_TurboGateValve_ILK(GEM1_PTM_30.iq_stPtm,GEM1_GPI_30.PG) AND GEM1_PTM_30.iq_stPtm.eState = pumpRUNNING,i_xOverrideMode := xGEM1OverrideMode);
 GEM1_VRC_50(i_xExtILK_OK := F_TurboGateValve_ILK(GEM1_PTM_50.iq_stPtm,GEM1_GPI_50.PG) AND GEM1_PTM_50.iq_stPtm.eState = pumpRUNNING,i_xOverrideMode := xGEM1OverrideMode);


(*Turbo vent valves NO*) //Deprecated
//GEM1_VVC_20(i_stPTM :=GEM1_PTM_20.iq_stPtm);
//GEM1_VVC_30(i_stPTM :=GEM1_PTM_30.iq_stPtm);
//GEM1_VVC_50(i_stPTM :=GEM1_PTM_50.iq_stPtm);
(*This part was added to Close all the Turbo's NO vent valves, These valves are capped off, and wont be in use*)
//GEM1_VVC_20.M_Close(TRUE);
//GEM1_VVC_10.M_Close(TRUE);
//GEM1_VVC_50.M_Close(TRUE);


(*Turbo Isolation valves*)
(*GEM1_PTM_10.i_xExtILKOk := F_TurboExtILK_NO(GEM1_PTM_10.iq_stPtm, GEM1_GPI_11.PG,
                        GEM1_GPI_10.PG,GEM1_VVC_20.q_stValve,GEM1_PRO_20.iq_stPFO);
GEM1_PTM_10(i_stGauge:=GEM1_GPI_11.PG,i_rMaxBackingPressure :=rMaxBackingPressure);*)
GEM1_PTM_10( i_xExtILKOk := F_TurboExtILKLogic_2(GEM1_PTM_10.iq_stPtm, GEM1_GPI_11.PG,
                        GEM1_GPI_10.PG,GEM1_PRO_20.iq_stPFO));
(*GEM1_PTM_20.i_xExtILKOk := F_TurboExtILK_NO(GEM1_PTM_20.iq_stPtm,BackingGauge:= GEM1_GPI_11.PG,
                        InletGauge:=GEM1_GPI_20.PG,GEM1_VVC_20.q_stValve,GEM1_PRO_20.iq_stPFO);
GEM1_PTM_20(i_stGauge:=GEM1_GPI_11.PG,i_rMaxBackingPressure :=rMaxBackingPressure);*)
GEM1_PTM_20( i_xExtILKOk := F_TurboExtILKLogic_2(GEM1_PTM_20.iq_stPtm, GEM1_GPI_11.PG,
                        GEM1_GPI_20.PG,GEM1_PRO_20.iq_stPFO));
GEM1_PTM_30(i_xExtILKOK:=F_TurboExtILKLogic_2(GEM1_PTM_30.iq_stPtm, GEM1_GPI_31.PG,
                        GEM1_GPI_30.PG,GEM1_PRO_30.iq_stPFO));
GEM1_PTM_50(i_xExtILKOK:=F_TurboExtILKLogic_2(GEM1_PTM_50.iq_stPtm, GEM1_GPI_51.PG,
                        GEM1_GPI_50.PG,GEM1_PRO_50.iq_stPFO));

(*Roughing pumps*)
GEM1_PRO_20(xExtIlk:= TRUE, TurboIsOn:= (GEM1_PTM_10.iq_stPtm.q_RunDO OR GEM1_PTM_20.iq_stPtm.q_RunDO));
GEM1_PRO_30(xExtIlk:= TRUE, TurboIsOn:= GEM1_PTM_30.iq_stPtm.q_RunDO);
GEM1_PRO_50(xExtIlk:= TRUE, TurboIsOn:= GEM1_PTM_50.iq_stPtm.q_RunDO);

END_PROGRAM

// ---- POUs/PRG_GEM2_DIFF_PUMP.TcPOU
PROGRAM PRG_GEM2_DIFF_PUMP
VAR
    rMaxBackingPressure : REAL := 0.7;
    bInit: BOOL:=TRUE;
END_VAR


(*Gauges*)
DSG_PIN(sNetId:='172.21.88.138.1.1' , nPort:=851 , sVarName:='GVL_Devices.AT2L0_SOLID_PIN_01',iWatchdog:=Main.iWatchdog,IG=> ); // Downstream Gauge from Down Stream PLC System
(*EM2L0*)
GEM2_GPI_30(PG=>);
GEM2_GCC_30(PG:=GEM2_GPI_30.PG,IG=>);
GEM2_GPI_31(PG=>);
GEM2_GPI_50(PG=>);
GEM2_GCC_50(PG:=GEM2_GPI_50.PG,IG=>);
GEM2_GPI_51(PG=>);
GEM2_GPI_60(PG=>);
GEM2_GCC_60(PG:=GEM2_GPI_60.PG,IG=>);
GEM2_GPI_61(PG=>);
GEM2_GPI_70(PG=>);
GEM2_GCC_70(PG:=GEM2_GPI_70.PG,IG=>);

(*VALVES*)
(*Aperture valve may open when Detector and Attenuator N2 valves are closed. Override provided *)
 (* to Include PMPS ILK with the EXTILK bit*)
(*apperture valves*)
GEM2_VGC_10(i_stUSG := GEM2_GPI_10.PG, i_stDSG:= GEM2_GPI_10.PG,i_xDis_DPIlk := TRUE, i_xEPS_OK := TRUE,
        i_xPMPS_OK := TRUE, i_xExt_OK := xGEM2_AperturesOpnOK, i_xOverrideMode := xGEM2OverrideMode,i_xReset := , i_xIsAperture:= TRUE ,
        io_fbFFHWO :=g_FastFaultOutput1,i_sDevName:= 'EM2L0:GEM:VGC:10',fbArbiter:=g_fbArbiter2,i_nTransitionRootID:=2100);
GEM2_VGC_20(i_stUSG := GEM2_GPI_10.PG, i_stDSG:= GEM2_GCC_30.IG,i_xDis_DPIlk := TRUE, i_xEPS_OK := TRUE,
        i_xPMPS_OK := TRUE, i_xExt_OK := xGEM2_AperturesOpnOK, i_xOverrideMode := xGEM2OverrideMode,i_xReset := , i_xIsAperture:= TRUE ,
        io_fbFFHWO :=g_FastFaultOutput1,i_sDevName:= 'EM2L0:GEM:VGC:20',fbArbiter:=g_fbArbiter2,i_nTransitionRootID:=2200);;
GEM2_VGC_30(i_stUSG := GEM2_GCC_30.IG, i_stDSG:= GEM2_GCC_30.IG,i_xDis_DPIlk := TRUE, i_xEPS_OK := TRUE,
        i_xPMPS_OK := TRUE, i_xExt_OK := xGEM2_AperturesOpnOK, i_xOverrideMode := xGEM2OverrideMode,i_xReset := , i_xIsAperture:= TRUE ,
        io_fbFFHWO :=g_FastFaultOutput1,i_sDevName:= 'EM2L0:GEM:VGC:30',fbArbiter:=g_fbArbiter2,i_nTransitionRootID:=2300);
GEM2_VGC_40(i_stUSG := GEM2_GCC_50.IG, i_stDSG:= GEM2_GCC_50.IG,i_xDis_DPIlk := TRUE, i_xEPS_OK := TRUE,
        i_xPMPS_OK := TRUE, i_xExt_OK := xGEM2_AperturesOpnOK, i_xOverrideMode := xGEM2OverrideMode,i_xReset := , i_xIsAperture:= TRUE ,
        io_fbFFHWO :=g_FastFaultOutput1,i_sDevName:= 'EM2L0:GEM:VGC:40',fbArbiter:=g_fbArbiter2,i_nTransitionRootID:=2400);
GEM2_VGC_50(i_stUSG := GEM2_GCC_30.IG, i_stDSG:= GEM2_GCC_60.IG,i_xDis_DPIlk := TRUE, i_xEPS_OK := TRUE,
        i_xPMPS_OK := TRUE, i_xExt_OK := xGEM2_AperturesOpnOK, i_xOverrideMode := xGEM2OverrideMode,i_xReset := , i_xIsAperture:= TRUE ,
        io_fbFFHWO :=g_FastFaultOutput1,i_sDevName:= 'EM2L0:GEM:VGC:50',fbArbiter:=g_fbArbiter2,i_nTransitionRootID:=2500);
GEM2_VGC_60(i_stUSG := GEM2_GCC_60.IG, i_stDSG:= GEM2_GCC_70.IG,i_xDis_DPIlk := TRUE, i_xEPS_OK := TRUE,
        i_xPMPS_OK := TRUE, i_xExt_OK := xGEM2_AperturesOpnOK, i_xOverrideMode := xGEM2OverrideMode,i_xReset := , i_xIsAperture:= TRUE ,
        io_fbFFHWO :=g_FastFaultOutput1,i_sDevName:= 'EM2L0:GEM:VGC:60',fbArbiter:=g_fbArbiter2,i_nTransitionRootID:=2600);
(*downstream isolation valve*)
GEM2_VGC_70(i_stUSG := GEM2_GCC_70.IG, i_stDSG:= DSG_PIN.IG,i_xDis_DPIlk := FALSE, i_xEPS_OK := TRUE,
        i_xPMPS_OK := TRUE, i_xExt_OK := NOT (DSG_PIN.bError) , i_xOverrideMode := xGEM2OverrideMode,i_xReset := ,
        io_fbFFHWO :=g_FastFaultOutput1,i_sDevName:= 'EM2L0:GEM:VGC:70',fbArbiter:=g_fbArbiter2,i_nTransitionRootID:=2700);
DSV_VGC(VGC=>);

(*Turbo vent valves NO*)//Deprecated
//GEM2_VVC_30(i_stPTM :=GEM2_PTM_30.iq_stPtm);
//GEM2_VVC_50(i_stPTM :=GEM2_PTM_50.iq_stPtm);
//GEM2_VVC_70(i_stPTM :=GEM2_PTM_70.iq_stPtm);
(*This part was added to Close all the Turbo's NO vent valves, These valves are capped off, and wont be in use*)
//GEM2_VVC_30.M_Close(TRUE);
//GEM2_VVC_50.M_Close(TRUE);
//GEM2_VVC_70.M_Close(TRUE);


(*Turbo Isolation valves*)
 GEM2_VRC_30(i_xExtILK_OK := F_TurboGateValve_ILK(GEM2_PTM_30.iq_stPtm,GEM2_GPI_30.PG) AND GEM2_PTM_30.iq_stPtm.eState = pumpRUNNING,i_xOverrideMode := xGEM2OverrideMode);
 GEM2_VRC_50(i_xExtILK_OK := F_TurboGateValve_ILK(GEM2_PTM_50.iq_stPtm,GEM2_GPI_50.PG) AND GEM2_PTM_50.iq_stPtm.eState = pumpRUNNING,i_xOverrideMode := xGEM2OverrideMode);
 GEM2_VRC_60(i_xExtILK_OK := F_TurboGateValve_ILK(GEM2_PTM_60.iq_stPtm,GEM2_GPI_60.PG) AND GEM2_PTM_60.iq_stPtm.eState = pumpRUNNING,i_xOverrideMode := xGEM2OverrideMode);
 GEM2_VRC_70(i_xExtILK_OK := F_TurboGateValve_ILK(GEM2_PTM_70.iq_stPtm,GEM2_GPI_70.PG) AND GEM2_PTM_70.iq_stPtm.eState = pumpRUNNING,i_xOverrideMode := xGEM2OverrideMode);

(*Turbo Pumps*)
GEM2_PTM_30(i_xExtILKOK:=F_TurboExtILKLogic_2(GEM2_PTM_30.iq_stPtm, GEM2_GPI_31.PG,
                        GEM2_GPI_30.PG,GEM2_PRO_30.iq_stPFO));
GEM2_PTM_50(i_xExtILKOK:=F_TurboExtILKLogic_2(GEM2_PTM_50.iq_stPtm, GEM2_GPI_51.PG,
                        GEM2_GPI_50.PG,GEM2_PRO_50.iq_stPFO));
GEM2_PTM_60(i_xExtILKOK:=F_TurboExtILKLogic_2(GEM2_PTM_60.iq_stPtm, GEM2_GPI_61.PG,
                        GEM2_GPI_60.PG,GEM2_PRO_60.iq_stPFO));
GEM2_PTM_70(i_xExtILKOK:=F_TurboExtILKLogic_2(GEM2_PTM_70.iq_stPtm, GEM2_GPI_61.PG,
                        GEM2_GPI_70.PG,GEM2_PRO_60.iq_stPFO));


(*Roughing pumps*)
GEM2_PRO_30(xExtIlk:= TRUE, TurboIsOn:= GEM2_PTM_30.iq_stPtm.q_RunDO);
GEM2_PRO_50(xExtIlk:= TRUE, TurboIsOn:= GEM2_PTM_50.iq_stPtm.q_RunDO);
GEM2_PRO_60(xExtIlk:= TRUE, TurboIsOn:= (GEM2_PTM_60.iq_stPtm.q_RunDO OR GEM2_PTM_70.iq_stPtm.q_RunDO));

END_PROGRAM

// ---- POUs/PRG_ROOTS.TcPOU
PROGRAM PRG_ROOTS
VAR
END_VAR

(*EM1L0*)
(*Roots Pump Chamber 1*)
(*gauges*)
GEM1_GPI_60(PG=>);
GEM1_GPI_61(PG=>);
GEM1_GPI_71(PG=>);

(*Isolation Valve*)
GEM1_VRC_60(Pump:=GEM1_PRO_60.q_stPump,Gauge:=GEM1_GPI_60.PG,i_xExtILK_OK:=TRUE);
GEM1_VRC_70(Pump:=GEM1_PRO_70.q_stPump,Gauge:=GEM1_GPI_60.PG,i_xExtILK_OK:=TRUE);


(* dry pump*)
GEM1_PRO_60();
GEM1_PRO_70();




(*EM2L0*)
(*Roots Pump Chamber 1*)
(*gauges*)
GEM2_GPI_10(PG=>);
GEM2_GPI_11(PG=>);
GEM2_GPI_21(PG=>);

(*Isolation Valve*)
GEM2_VRC_10(Pump:=GEM2_PRO_10.q_stPump,Gauge:=GEM2_GPI_10.PG,i_xExtILK_OK:=TRUE);
GEM2_VRC_20(Pump:=GEM2_PRO_20.q_stPump,Gauge:=GEM2_GPI_10.PG,i_xExtILK_OK:=TRUE);

(* dry pump*)
GEM2_PRO_10();
GEM2_PRO_20();

END_PROGRAM

// ---- POUs/PRG_GATT.TcPOU
PROGRAM PRG_GATT
VAR CONSTANT
        nDataTable_NumberOfRows : INT:=9;
END_VAR
VAR
    (*needle valve control position*)
    VCN_Req_Pos: REAL;

    fb_PID: FB_BasicPID;

    {attribute 'pytmc' :=' pv: AT1L0:GAS:CNTRL:SP '}
    fSetpointValue : REAL:=0.001;
    {attribute 'pytmc' :=' pv: AT1L0:GAS:CNTRL:Kp '}
    fKp : REAL:= 1.1;
    {attribute 'pytmc' :=' pv: AT1L0:GAS:CNTRL:Tn '}
    fTn : REAL:= 0.5;




    eMode							: E_CTRL_MODE;
    stCTRL_PID_PARAMS		: ST_CTRL_PID_PARAMS;

    eErrorId						: E_CTRL_ERRORCODES;
    bError							: BOOL;
    bARWactive					: BOOL;

    (* controller *)
    fbCTRL_PID					: FB_CTRL_PID;
    bInit							: BOOL	:= TRUE;

    stCTRL_LIN_INTERPOLATION_PARAMS		: ST_CTRL_LIN_INTERPOLATION_PARAMS;
    arrTable											: ARRAY[1..nDataTable_NumberOfRows,1..2] OF FLOAT;

END_VAR

(*Gauges*)
GATT_GPI_10();
GATT_GMP_10(i_rFULL_SCALE := 2.0 (*Torr*));
GATT_GMP_11();

(*Valves*)
(*Gas Cell vent valve*)
GATT_VRC_10(i_xExtILK_OK:= GEM2_VGC_70.iq_stValve.i_xClsLS AND DSV_VGC.VGC.i_xClsLS AND GEM1_Turbo_Valves_Closed AND GEM2_Turbo_Valves_Closed AND TwinscrewPumps_Valves_Closed, i_xOverrideMode := xGATTOverrideMode);

(* N2 Cutt off valve*)
GATT_VVC_10(i_xExtILK_OK := GEM1_Aperture_Closed AND GEM1_Turbo_Valves_Open AND GEM1_Turbo_Running AND GEM2_Aperture_Closed AND GEM2_Turbo_Valves_Open AND GEM2_Turbo_Running AND GEM1_TwinscrewPumps_Valves_Open AND GEM2_TwinscrewPumps_Valves_Open);

END_PROGRAM

// ---- POUs/PRG_GEM1.TcPOU
PROGRAM PRG_GEM1
VAR
    {attribute 'pytmc' :=' pv: EM1L0:GEM:CNTRL:RESET;
     field: ZNAM FALSE;
     field: ONAM TRUE;
     io: io;
    '}
    bReset : BOOL;
    {attribute 'pytmc' :=' pv: EM1L0:GEM:CNTRL:ERROR;
     field: ZNAM FALSE;
     field: ONAM TRUE;
     io: io;
    '}
    bError : BOOL;
    {attribute 'pytmc' :=' pv: EM1L0:GEM:CNTRL:Kp1 '}
    fKp1 : REAL:= 0.4;
    {attribute 'pytmc' :=' pv: EM1L0:GEM:CNTRL:Tn1 '}
    fTn1 : REAL:= 0.5;
    {attribute 'pytmc' :=' pv: EM1L0:GEM:CNTRL:Kp2 '}
    fKp2 : REAL:= 0.01;
    {attribute 'pytmc' :=' pv: EM1L0:GEM:CNTRL:Tn2 '}
    fTn2 : REAL:= 0.5;
    arrTable_GEM1	: ARRAY[1..30,1..2] OF FLOAT;
    fManValue											: FLOAT;
    bExtrapolate										: BOOL;
    eMode							: E_CTRL_MODE;
    stCTRL_PID_PARAMS		: ST_CTRL_PID_PARAMS;
    bSync							: BOOL;
    bHold							: BOOL;
    eErrorId						: E_CTRL_ERRORCODES;
    bARWactive					: BOOL;
    (* controller *)
    fbCTRL_PID					: FB_CTRL_PID;
    bInit							: BOOL	:= TRUE;
    fbCTRL_LIN_INTERPOLATION					: FB_CTRL_LIN_INTERPOLATION;
    //stCTRL_LIN_INTERPOLATION_PARAMS		: ST_CTRL_LIN_INTERPOLATION_PARAMS;
    stCTRL_LIN_INTERPOLATION_PARAMS_GEM	: ST_CTRL_LIN_INTERPOLATION_PARAMS;
    fbCTRL_DEADBAND						: FB_CTRL_DEADBAND;
    stCTRL_DEADBAND_PARAMS			: ST_CTRL_DEADBAND_PARAMS;
        //timer to switch the pid from manual to active 5seconds??? 10 seconds???
    pid_on :TON;
    wait : time := T#10S;
FTrig: F_TRIG;


END_VAR


(*Devices*)
(* GEM 1*)
(*Gauges*)
GEM1_GCM_41(i_rFULL_SCALE := 10.0 (*Torr*));
GEM1_GCM_42(i_rFULL_SCALE := 0.05 (*Torr*));
(*Assign reading to psuedo gauge*)
IF (GEM1_GCM_42.PG.rPRESS >=0.049) THEN GEM1_GCM_40 := GEM1_GCM_41.PG;
    ELSE
    GEM1_GCM_40 := GEM1_GCM_42.PG;
END_IF
(* Gauge selection *)
fbCTRL_PID.fActualValue := GEM1_GCM_40.rPRESS;
(*
IF (fGEM1SetpointValue >=0.049) THEN
    fbCTRL_PID.fActualValue := GEM1_GCM_41.PG.rPRESS;
ELSE
    fbCTRL_PID.fActualValue := GEM1_GCM_42.PG.rPRESS;
END_IF*)


(* N2 Cut Off Valves *)
GEM1_VVC_40(i_xExtILK_OK:= GEM1_Aperture_Closed AND GEM1_Turbo_Valves_Open AND GEM1_Turbo_Running);

(*Flow Control Valves*)
GEM1_VCN_40 (i_xExtIlkOK := (GEM1_Aperture_Closed AND GEM1_Turbo_Valves_Open AND GEM1_Turbo_Running),// AND  GEM1_VVC_40.M_IsOpen()),
             i_ReqPos:= fbCTRL_LIN_INTERPOLATION.fOut + fbCTRL_PID.fOut);
//GEM1_VPC_42 (i_xExtIlkOK := TRUE, i_rReqPos:= );



(*Iniitialization*)
IF bInit
THEN


    (* init array with the interpolation points  *)
    (* 	fIn					 |		fOut		*)
    arrTable_GEM1[1,1] := 0;		arrTable_GEM1[1,2] := 23.8;
    arrTable_GEM1[2,1] := 0.00178;		arrTable_GEM1[2,2] := 23.9;
    arrTable_GEM1[3,1] := 0.0025;		arrTable_GEM1[3,2] := 24;
    arrTable_GEM1[4,1] :=  0.005884;	    arrTable_GEM1[4,2] := 25;
    arrTable_GEM1[5,1] :=  0.085;	    arrTable_GEM1[5,2] := 35;
    arrTable_GEM1[6,1] := 0.1263;		arrTable_GEM1[6,2] := 40;
    arrTable_GEM1[7,1] := 0.1626;		arrTable_GEM1[7,2] := 42;
    arrTable_GEM1[8,1] := 0.19;	    arrTable_GEM1[8,2] := 44;
    arrTable_GEM1[9,1] := 0.234;	    arrTable_GEM1[9,2] := 46;
    arrTable_GEM1[10,1] := 0.32;		arrTable_GEM1[10,2] := 50;
    arrTable_GEM1[11,1] := 0.370;		arrTable_GEM1[11,2] := 52;
    arrTable_GEM1[12,1] := 0.43427;		arrTable_GEM1[12,2] := 54;
    arrTable_GEM1[13,1] := 0.5316;		arrTable_GEM1[13,2] := 55;
    arrTable_GEM1[14,1] := 0.61;		arrTable_GEM1[14,2] := 55.5;
    arrTable_GEM1[15,1] := 0.894;		arrTable_GEM1[15,2] := 56;
    arrTable_GEM1[16,1] := 1.215;		arrTable_GEM1[16,2] := 56.5;
    arrTable_GEM1[17,1] := 1.58;		arrTable_GEM1[17,2] := 57;
    arrTable_GEM1[18,1] := 2.025;	    arrTable_GEM1[18,2] := 58;
    arrTable_GEM1[19,1] := 2.2;	    arrTable_GEM1[19,2] :=58.1;
    arrTable_GEM1[20,1] := 2.9;		arrTable_GEM1[20,2] := 65;
    arrTable_GEM1[21,1] := 3;		arrTable_GEM1[21,2] := 69;
    arrTable_GEM1[22,1] :=  3.0448;	    arrTable_GEM1[22,2] := 70;
    arrTable_GEM1[23,1] :=  3.31919;	    arrTable_GEM1[23,2] := 72;
    arrTable_GEM1[24,1] :=3.324;		arrTable_GEM1[24,2] := 73.04;
    arrTable_GEM1[25,1] :=3.71941;		arrTable_GEM1[25,2] := 73.64;
    arrTable_GEM1[26,1] := 3.81941;		arrTable_GEM1[26,2] := 74.45;
    arrTable_GEM1[27,1] :=  3.963194;		arrTable_GEM1[27,2] :=74.46;
    arrTable_GEM1[28,1] := 3.99999;	arrTable_GEM1[28,2] := 75;
    arrTable_GEM1[29,1] :=  4;		arrTable_GEM1[29,2] :=75.5;
    arrTable_GEM1[30,1] := 4.1;	arrTable_GEM1[30,2] := 75.505;

    (* init parameter struct *)
    stCTRL_LIN_INTERPOLATION_PARAMS_GEM.tCtrlCycleTime					:= T#10ms;
    stCTRL_LIN_INTERPOLATION_PARAMS_GEM.tTaskCycleTime					:= T#10ms;
    stCTRL_LIN_INTERPOLATION_PARAMS_GEM.nDataTable_NumberOfRows		:= INT_TO_UINT(30);


    (* init parameter struct *)
    stCTRL_PID_PARAMS.tCtrlCycleTime		:= T#10ms;
    stCTRL_PID_PARAMS.tTaskCycleTime		:= T#10ms;
    stCTRL_PID_PARAMS.fKp					:= fKp1;			(* proportional gain Kp				*)
    stCTRL_PID_PARAMS.tTn					:= T#1s;		(*  Tn									*)
    stCTRL_PID_PARAMS.tTv					:= T#200ms;	(*  Tv									*)
    stCTRL_PID_PARAMS.tTd					:= T#200ms;	(*  Td									*)
    stCTRL_PID_PARAMS.fOutMaxLimit			:=  5;			(* maximum output limit				*)
    stCTRL_PID_PARAMS.fOutMinLimit			:=  -100;			(* minimum output limit				*)

    (* set the mode to ACTIVE --> normal operation *)
    eMode							:= eCTRL_MODE_PASSIVE    ;
    (* reset the init flag *)
    bInit							:= FALSE;
END_IF
(* set the addresses *)
stCTRL_LIN_INTERPOLATION_PARAMS_GEM.pDataTable_ADR			:= ADR(arrTable_GEM1);
stCTRL_LIN_INTERPOLATION_PARAMS_GEM.nDataTable_SIZEOF		:= SIZEOF(arrTable_GEM1);


